(* IEC 61131-3 sources: manufacturing_io/scenes, 18 files *)

(* ---- a-to-b.st ---- *)
VAR
	START_EDGE : BOOL;
	PB_START_LAST : BOOL;
	STOP_REQ : BOOL;
	SEL_LAST : BOOL := TRUE;
	SEL_CHANGED : BOOL;
	T_DWELL : TON;
	T_WD : TON;
	EM_LAST : UDINT;
	STEP_LAST : UDINT;
	GONE : UDINT;
	MEM_CV : BOOL;
	IND_CV_LAST : BOOL;
	ESTOP : BOOL;
	READY : BOOL;
	MASTER_ON : BOOL;
	HOMED : BOOL;
	MASTER_EDGE : BOOL;
	PB_MASTER_LAST : BOOL;
	HOME_EDGE : BOOL;
	PB_HOME_LAST : BOOL;
END_VAR
// a-to-b: load one part, carry it to the end sensor, dwell, discharge it to the unloader, repeat
// until STOP. The same sequence runs without a PLC in a-to-b.ctl.js.
//
// Waiting steps wait for an INVARIANT, not for a counter to move: a change cannot say which
// part moved (measured on the simulator: parts piled up, then pipelined).
//
// The panel has a selector AUTO / INDIVIDUAL (rb4axis): START only in AUTO, the individual buttons
// only in INDIVIDUAL, and a change while the sequence runs is a FAULT, not a pause.

START_EDGE := PB_START AND NOT PB_START_LAST;
PB_START_LAST := PB_START;
IF PB_CSTOP THEN
	STOP_REQ := TRUE;
END_IF;
SEL_CHANGED := SEL_AUTO <> SEL_LAST;
SEL_LAST := SEL_AUTO;

// The master circuit, as on the cell panel: E-STOP is a latching mushroom, MASTER ON energises
// the machine, and nothing runs without it. An E-STOP also loses the home position.
ESTOP := PB_ESTOP;
MASTER_EDGE := PB_MASTER AND NOT PB_MASTER_LAST;
PB_MASTER_LAST := PB_MASTER;
HOME_EDGE := PB_HOME AND NOT PB_HOME_LAST;
PB_HOME_LAST := PB_HOME;
IF ESTOP THEN
	MASTER_ON := FALSE;
	HOMED := FALSE;
ELSIF MASTER_EDGE THEN
	MASTER_ON := TRUE;
END_IF;
READY := MASTER_ON AND NOT ESTOP;

// A write-off goes STALE when the part turns up after all - the hand puts it back, or it reaches
// the unloader later. Then RM + GONE runs PAST EM and step 40 stops waiting at all. GONE is a
// UDINT, so EM1_CNT - RM1_CNT with RM ahead underflows to about 4 billion: guard before you
// subtract.
IF RM1_CNT >= EM1_CNT THEN
	GONE := 0;
ELSIF RM1_CNT + GONE > EM1_CNT THEN
	GONE := EM1_CNT - RM1_CNT;
END_IF;

CASE ST1_STEP OF
	0:	// idle
		CV1_RUN := FALSE;
		EM1_EMIT := FALSE;
		IF START_EDGE AND SEL_AUTO AND READY AND HOMED THEN
			STOP_REQ := FALSE;
			EM_LAST := EM1_CNT;
			ST1_STEP := 10;
		END_IF;
	10:	// load one part: the command is held until the loader's counter answers it
		EM1_EMIT := TRUE;
		IF EM1_CNT <> EM_LAST THEN
			EM1_EMIT := FALSE;
			ST1_STEP := 15;
		END_IF;
	15:	// the beam must be clear before this part runs to it
		CV1_RUN := TRUE;
		IF NOT PE_END THEN
			ST1_STEP := 20;
		END_IF;
	20:	// carry it to the end sensor
		CV1_RUN := TRUE;
		IF PE_END THEN
			CV1_RUN := FALSE;
			ST1_STEP := 30;
		END_IF;
	30:	// dwell
		IF T_DWELL.Q THEN
			ST1_STEP := 40;
		END_IF;
	40:	// discharge: every part loaded has left the belt (counting the write-offs)
		CV1_RUN := TRUE;
		IF RM1_CNT + GONE >= EM1_CNT THEN
			CV1_RUN := FALSE;
			ST1_STEP := 50;
		END_IF;
	50:	// cycle complete
		CYCLE_CNT := CYCLE_CNT + 1;
		IF STOP_REQ THEN
			ST1_STEP := 0;
		ELSE
			EM_LAST := EM1_CNT;
			ST1_STEP := 10;
		END_IF;
	800:	// HOME: nothing here is positioned, so home only has to leave the line quiet
		CV1_RUN := FALSE;
		EM1_EMIT := FALSE;
		HOMED := TRUE;
		ST1_STEP := 0;
	910:	// E-STOP: the master circuit is open, so every solenoid de-energises - which is what
		// really happens: a 5/2 single-solenoid valve springs back, a double one holds.
		CV1_RUN := FALSE;
		EM1_EMIT := FALSE;
		IF READY THEN	// MASTER ON after the mushroom is released
			ST1_STEP := 0;
		END_IF;
	900:	// FAULT: a step stopped moving. Hold everything until START acknowledges it.
		CV1_RUN := FALSE;
		EM1_EMIT := FALSE;
		IF START_EDGE AND SEL_AUTO THEN
			STOP_REQ := FALSE;
			// Acknowledging writes off whatever never reached the unloader. Only HERE: at every
			// START it would write off parts still legitimately on the belt, and then an older
			// part's removal ends this cycle - the pipelining bug that cost two live rounds.
			GONE := EM1_CNT - RM1_CNT;
			ST1_STEP := 0;
		END_IF;
END_CASE;

T_DWELL(In := (ST1_STEP = 30), PT := T#500ms);

// Watchdog: a running step that stops moving is a jam, not patience. A selector change while
// running trips the same way.
T_WD(In := (ST1_STEP = STEP_LAST) AND (ST1_STEP <> 0) AND (ST1_STEP <> 900) AND (ST1_STEP <> 910), PT := T#15s);
IF ST1_STEP <> STEP_LAST THEN
	STEP_LAST := ST1_STEP;
END_IF;
IF T_WD.Q OR (SEL_CHANGED AND (ST1_STEP <> 0) AND (ST1_STEP <> 900) AND (ST1_STEP <> 910)) THEN
	ST1_STEP := 900;
	CV1_RUN := FALSE;
	EM1_EMIT := FALSE;
END_IF;

// E-STOP at any moment, and the HOME button when the machine is energised and idle.
IF ESTOP THEN
	IF ST1_STEP <> 910 THEN
		ST1_STEP := 910;
	END_IF;
	CV1_RUN := FALSE;
	EM1_EMIT := FALSE;
ELSIF HOME_EDGE AND READY AND (ST1_STEP = 0) THEN
	ST1_STEP := 800;
END_IF;

AUTO_RUN := (ST1_STEP <> 0) AND (ST1_STEP <> 800) AND (ST1_STEP <> 900) AND (ST1_STEP <> 910);

// Individual operation: the buttons are momentary; the PLC keeps a toggle
// memory per actuator and clears it when INDIVIDUAL ends, so nothing stays latched into AUTO.
IF NOT SEL_AUTO AND NOT AUTO_RUN AND READY AND (ST1_STEP <> 800) THEN
	IF IND_CV AND NOT IND_CV_LAST THEN
		MEM_CV := NOT MEM_CV;
	END_IF;
	CV1_RUN := MEM_CV;
	EM1_EMIT := IND_FEED;
ELSE
	MEM_CV := FALSE;
END_IF;
IND_CV_LAST := IND_CV;

// The speed override the operator dialled in, passed on to the axes and the belts.
OVR := OVR_SET;

PL_START := AUTO_RUN;
PL_MASTER := MASTER_ON;
PL_HOME := HOMED;

(* ---- assembler.st ---- *)
VAR
	START_EDGE : BOOL;
	PB_START_LAST : BOOL;
	STOP_REQ : BOOL;
	EM_B_LAST : UDINT;
	EM_L_LAST : UDINT;
	NEXT_ST : INT;
	T_PRESS : TON;
END_VAR
// assembler: a 4-station cam indexer. Every station works during the same dwell - load a base,
// drop a lid on it, press it - and then the table turns one step, carrying each assembly to the
// next station. The unload station simply takes whatever reaches it. The same sequence runs
// without a PLC in assembler.ctl.js.
//
// The index waits for an INVARIANT, TBL_STATION = NEXT_ST, not for the station to change: a
// change cannot say which index it belonged to, and OPC UA sampling can miss a short state.
// Each feeder command is held until that feeder's own counter answers it.

START_EDGE := PB_START AND NOT PB_START_LAST;
PB_START_LAST := PB_START;
IF PB_STOP THEN
	STOP_REQ := TRUE;
END_IF;

CASE ST1_STEP OF
	0:	// idle, table stopped in a dwell, press up
		TBL_RUN := FALSE;
		EM_B_EMIT := FALSE;
		EM_L_EMIT := FALSE;
		SOL_PRESS_DN := FALSE;
		SOL_PRESS_UP := TRUE;
		IF START_EDGE AND TBL_INPOS AND AS_PRESS_UP THEN
			STOP_REQ := FALSE;
			EM_B_LAST := EM_B_CNT;
			ST1_STEP := 10;
		END_IF;
	10:	// station 0: load a base into the nest
		EM_B_EMIT := TRUE;
		IF EM_B_CNT <> EM_B_LAST THEN
			EM_B_EMIT := FALSE;
			EM_L_LAST := EM_L_CNT;
			ST1_STEP := 20;
		END_IF;
	20:	// station 1: drop a lid onto the base that arrived there
		EM_L_EMIT := TRUE;
		IF EM_L_CNT <> EM_L_LAST THEN
			EM_L_EMIT := FALSE;
			ST1_STEP := 30;
		END_IF;
	30:	// station 2: press down
		SOL_PRESS_UP := FALSE;
		SOL_PRESS_DN := TRUE;
		IF AS_PRESS_DN THEN
			ST1_STEP := 40;
		END_IF;
	40:	// hold the press on the lid
		IF T_PRESS.Q THEN
			ST1_STEP := 50;
		END_IF;
	50:	// press up, and pick the station this index must reach
		SOL_PRESS_DN := FALSE;
		SOL_PRESS_UP := TRUE;
		IF AS_PRESS_UP THEN
			NEXT_ST := (TBL_STATION + 1) MOD 4;
			ST1_STEP := 60;
		END_IF;
	60:	// turn the table one station
		TBL_RUN := TRUE;
		IF TBL_INPOS AND TBL_STATION = NEXT_ST THEN
			TBL_RUN := FALSE;
			CYCLE_CNT := CYCLE_CNT + 1;
			IF STOP_REQ THEN
				ST1_STEP := 0;
			ELSE
				EM_B_LAST := EM_B_CNT;
				ST1_STEP := 10;
			END_IF;
		END_IF;
END_CASE;

T_PRESS(In := (ST1_STEP = 40), PT := T#300ms);
AUTO_RUN := ST1_STEP <> 0;
PL_START := AUTO_RUN;

(* ---- blurobot.st ---- *)
VAR
	START_EDGE : BOOL;
	PB_START_LAST : BOOL;
	STOP_REQ : BOOL;
	T_WD : TON;
	T_GRIP : TON;
	STEP_LAST : UDINT;
	i : INT;
	j : INT;
	SRC : INT;
	DST : INT;
	IDX : INT;
	HOLDING : BOOL;
	AT_POSE : BOOL;
	CLEARED : BOOL;
	RAIL_X : LREAL;
	ARM_AT_1 : LREAL;
	ARM_AT_2 : LREAL;
	ARM_AT_3 : LREAL;
	ARM_UP_1 : LREAL;
	ARM_UP_2 : LREAL;
	ARM_UP_3 : LREAL;
	COVER_OK : BOOL;
	IN_ZONE : BOOL;
	SHUT : BOOL;
	// What the PLC BELIEVES about each station, and each machine's own clock. These are program
	// variables, not machine IO: nothing in the plant senses them. rb4axis keeps the same values in
	// SIM_ST_STATE / SIM_ST_TIMER and only publishes them so its viewer can draw the cell.
	//   0 empty, 1 processing, 2 finished and waiting to be collected
	ICC1_STATE : INT;
	ICC2_STATE : INT;
	DW1_STATE : INT;
	DW2_STATE : INT;
	ICC1_TIMER : LREAL;
	ICC2_TIMER : LREAL;
	DW1_TIMER : LREAL;
	DW2_TIMER : LREAL;
	// The cover target each station is latched on. Execute is LATCHED on its rising edge, like
	// every other axis here, so holding it true from the first scan means the target is never
	// re-read: measured, the covers held their startup 80 while the target sat at 0, no ICC clock
	// ever ran, and no board ever finished. A change re-pulses Execute.
	ICC1_CV_WANT : LREAL;
	ICC2_CV_WANT : LREAL;
	DW1_CV_WANT : LREAL;
	DW2_CV_WANT : LREAL;
END_VAR
// blurobot - a PORT of rb4axis PRG_SIM_ROBOT.st. The cell, the station table, the job priorities,
// the step numbers and the timings are that program's; only the tag shape differs, because this
// repo binds scalar tags while the original keeps SIM_ST_* arrays.
//
//   station   type  rail x   surface z   process
//   WIP IN     0     -1400      250        -      stock is not simulated: always FULL
//   ICC 1      1      -700      285      17.0 s   test; the cover presses the PCB onto the probes
//   ICC 2      1      -300      285      17.0 s
//   DW 1       2       300      250      15.0 s   data writer
//   DW 2       2       700      250      15.0 s
//   WIP OUT    3      1400      250        -      the product leaves: always EMPTY
//
// Job priority, and the ORDER is the behaviour:
//   1. fill an EMPTY ICC from WIP IN - both - before anything else. That is what buffer means: the
//      17 s tester must not idle while the robot runs errands for DW.
//   2. empty a FINISHED DW to WIP OUT, ahead of 3, so a free DW always exists. Without it two full
//      DWs plus two finished ICCs deadlock, and the deadlock looks like a robot that stopped.
//   3. move a FINISHED ICC to an EMPTY DW.
//
// Poses were measured against the scene's own kinematics with the carriage at z 200: all twelve
// (six surfaces + six 140 mm approaches) solve with 67.3 deg of worst-case joint margin. Only two
// station heights exist, so there are four arm poses and the rail carries the difference.
//
// Execute is a LEVEL held until every axis reports Done, and the next move waits for Done to fall
// again: a one-scan pulse falls between two OPC UA samples.

START_EDGE := PB_START AND NOT PB_START_LAST;
PB_START_LAST := PB_START;
IF PB_STOP THEN
	STOP_REQ := TRUE;
END_IF;

AT_POSE := A0_DONE AND A1_DONE AND A2_DONE AND A3_DONE;
CLEARED := NOT A0_DONE AND NOT A1_DONE AND NOT A2_DONE AND NOT A3_DONE;

// ---------------------------------------------------------------- the machines
// Each keeps its OWN timer, running together: that is the whole point of a buffer, ICC 1 and ICC 2
// must be able to test at the same time while the robot is away. The clock runs ONLY with the
// cover shut - the cover presses the PCB onto the probes, and counting before it closes means
// claiming a test on a board nothing has touched.
//
// The cover closes only while processing and REOPENS if the arm is in its sweep: a light curtain,
// not a delay. Without it the leaf swings onto an arm that is still lifting out.
IN_ZONE := (ABS(A0_POS - (-700.0)) < 200.0) AND (A1_POS < 60.0);
SHUT := (ICC1_STATE = 1) AND NOT IN_ZONE;
IF SHUT THEN COVER_TARGET := 0.0; ELSE COVER_TARGET := 80.0; END_IF;
IF COVER_TARGET <> ICC1_CV_WANT THEN
	ICC1_CV_WANT := COVER_TARGET;
	ICC1_CV_EXEC := FALSE;
ELSE
	ICC1_CV_TGT := COVER_TARGET;
	ICC1_CV_EXEC := TRUE;
END_IF;
IF (ICC1_STATE = 1) AND (ICC1_CV_POS <= 0.5) THEN
	ICC1_TIMER := ICC1_TIMER - 0.002;
	IF ICC1_TIMER <= 0.0 THEN ICC1_TIMER := 0.0; ICC1_STATE := 2; END_IF;
END_IF;

IN_ZONE := (ABS(A0_POS - (-300.0)) < 200.0) AND (A1_POS < 60.0);
SHUT := (ICC2_STATE = 1) AND NOT IN_ZONE;
IF SHUT THEN COVER_TARGET := 0.0; ELSE COVER_TARGET := 80.0; END_IF;
IF COVER_TARGET <> ICC2_CV_WANT THEN
	ICC2_CV_WANT := COVER_TARGET;
	ICC2_CV_EXEC := FALSE;
ELSE
	ICC2_CV_TGT := COVER_TARGET;
	ICC2_CV_EXEC := TRUE;
END_IF;
IF (ICC2_STATE = 1) AND (ICC2_CV_POS <= 0.5) THEN
	ICC2_TIMER := ICC2_TIMER - 0.002;
	IF ICC2_TIMER <= 0.0 THEN ICC2_TIMER := 0.0; ICC2_STATE := 2; END_IF;
END_IF;

IN_ZONE := (ABS(A0_POS - 300.0) < 200.0) AND (A1_POS < 60.0);
SHUT := (DW1_STATE = 1) AND NOT IN_ZONE;
IF SHUT THEN COVER_TARGET := 0.0; ELSE COVER_TARGET := 80.0; END_IF;
IF COVER_TARGET <> DW1_CV_WANT THEN
	DW1_CV_WANT := COVER_TARGET;
	DW1_CV_EXEC := FALSE;
ELSE
	DW1_CV_TGT := COVER_TARGET;
	DW1_CV_EXEC := TRUE;
END_IF;
IF (DW1_STATE = 1) AND (DW1_CV_POS <= 0.5) THEN
	DW1_TIMER := DW1_TIMER - 0.002;
	IF DW1_TIMER <= 0.0 THEN DW1_TIMER := 0.0; DW1_STATE := 2; END_IF;
END_IF;

IN_ZONE := (ABS(A0_POS - 700.0) < 200.0) AND (A1_POS < 60.0);
SHUT := (DW2_STATE = 1) AND NOT IN_ZONE;
IF SHUT THEN COVER_TARGET := 0.0; ELSE COVER_TARGET := 80.0; END_IF;
IF COVER_TARGET <> DW2_CV_WANT THEN
	DW2_CV_WANT := COVER_TARGET;
	DW2_CV_EXEC := FALSE;
ELSE
	DW2_CV_TGT := COVER_TARGET;
	DW2_CV_EXEC := TRUE;
END_IF;
IF (DW2_STATE = 1) AND (DW2_CV_POS <= 0.5) THEN
	DW2_TIMER := DW2_TIMER - 0.002;
	IF DW2_TIMER <= 0.0 THEN DW2_TIMER := 0.0; DW2_STATE := 2; END_IF;
END_IF;

// WIP IN never runs out and WIP OUT never fills up: the stock either side of the cell is not
// simulated, and pretending otherwise would starve or block a cell that never does either. Those
// two need no state variable at all - the job selection below simply treats them that way.

// ---------------------------------------------------------- the pose for IDX
// Four arm poses only, because the six stations sit at just two heights; the rail carries the
// rest. Measured against the scene's own kinematics with the carriage at z 200.
CASE IDX OF
	0:	RAIL_X := -1400.0;
	1:	RAIL_X := -700.0;
	2:	RAIL_X := -300.0;
	3:	RAIL_X := 300.0;
	4:	RAIL_X := 700.0;
	5:	RAIL_X := 1400.0;
ELSE
	RAIL_X := 0.0;
END_CASE;

IF (IDX = 1) OR (IDX = 2) THEN
	// the 285 mm tables
	ARM_AT_1 := 15.72;   ARM_AT_2 := -71.33;   ARM_AT_3 := -34.39;
	ARM_UP_1 := 36.55;   ARM_UP_2 := -77.44;   ARM_UP_3 := -49.11;
ELSE
	// the 250 mm tables
	ARM_AT_1 := 9.76;   ARM_AT_2 := -67.25;   ARM_AT_3 := -32.5;
	ARM_UP_1 := 31.86;   ARM_UP_2 := -77.37;   ARM_UP_3 := -44.49;
END_IF;

// The WIP racks are open - no cover, so nothing to wait for.
CASE IDX OF
	1:	COVER_OK := ICC1_CV_POS >= 79.5;
	2:	COVER_OK := ICC2_CV_POS >= 79.5;
	3:	COVER_OK := DW1_CV_POS >= 79.5;
	4:	COVER_OK := DW2_CV_POS >= 79.5;
ELSE
	COVER_OK := TRUE;
END_CASE;

// ------------------------------------------------- every station holds what is on it
// Only the one being picked from lets go, and only while the gripper takes the board. Measured
// with no clamp set at all: the nest held nothing, WIPIN_P never came true, and the fingers closed
// to zero straight through the PCB - a part's width is only measured for a FREE part, so gripping
// a still-held board reads as gripping air and the closed switch asserts for the wrong reason.
// WIP IN is an ENDLESS stock: the PLC pins its state to "full" because the racks either side of
// the cell are not simulated, so the plant has to keep a board there or the cell runs dry and the
// next grip closes on air. A LEVEL held until the feeder's own count answers it, never a pulse,
// and only while that nest is empty and the arm is not taking from it.
EM_IN_EMIT := NOT WIPIN_P AND NOT (((ST1_STEP = 14) OR (ST1_STEP = 15)) AND (IDX = 0));

WIPIN_CLAMP := NOT (((ST1_STEP = 14) OR (ST1_STEP = 15)) AND (IDX = 0));
ICC1_CLAMP := NOT (((ST1_STEP = 14) OR (ST1_STEP = 15)) AND (IDX = 1));
ICC2_CLAMP := NOT (((ST1_STEP = 14) OR (ST1_STEP = 15)) AND (IDX = 2));
DW1_CLAMP := NOT (((ST1_STEP = 14) OR (ST1_STEP = 15)) AND (IDX = 3));
DW2_CLAMP := NOT (((ST1_STEP = 14) OR (ST1_STEP = 15)) AND (IDX = 4));
WIPOUT_CLAMP := NOT (((ST1_STEP = 14) OR (ST1_STEP = 15)) AND (IDX = 5));

CASE ST1_STEP OF
	0:	// pick a job - the order of these three searches IS the cell's behaviour
		SRC := -1;
		DST := -1;
		IF (ICC1_STATE = 0) THEN SRC := 0; DST := 1; END_IF;
		IF (DST < 0) AND (ICC2_STATE = 0) THEN SRC := 0; DST := 2; END_IF;
		IF (DST < 0) AND (DW1_STATE = 2) THEN SRC := 3; DST := 5; END_IF;
		IF (DST < 0) AND (DW2_STATE = 2) THEN SRC := 4; DST := 5; END_IF;
		IF (DST < 0) AND (ICC1_STATE = 2) AND (DW1_STATE = 0) THEN SRC := 1; DST := 3; END_IF;
		IF (DST < 0) AND (ICC1_STATE = 2) AND (DW2_STATE = 0) THEN SRC := 1; DST := 4; END_IF;
		IF (DST < 0) AND (ICC2_STATE = 2) AND (DW1_STATE = 0) THEN SRC := 2; DST := 3; END_IF;
		IF (DST < 0) AND (ICC2_STATE = 2) AND (DW2_STATE = 0) THEN SRC := 2; DST := 4; END_IF;
		IF DST >= 0 THEN
			IDX := SRC;
			ST1_STEP := 5;
		ELSIF STOP_REQ THEN
			STOP_REQ := FALSE;
		END_IF;

	5:	// fold to the travel pose - axes 1-3 only, the rail is not touched
		A1_TGT := 90.0;   A2_TGT := -90.0;   A3_TGT := -90.0;
		A1_EXEC := TRUE;   A2_EXEC := TRUE;   A3_EXEC := TRUE;
		IF A1_DONE AND A2_DONE AND A3_DONE THEN
			ST1_STEP := 7;
		END_IF;

	7:	// slide the rail. The arm MUST be folded: travelling while reaching down sweeps every
		// machine it passes, and on screen that looks perfectly smooth.
		A0_TGT := RAIL_X;
		A0_EXEC := TRUE;
		ST1_STEP := 8;

	8:	// TWO things, and the wait is HERE rather than after the approach is asked for: asking
		// while the cover is still shut gets the move refused, nothing moves, and Done stays TRUE -
		// so the next step would drive straight down from the travel pose, skipping the approach.
		IF A0_DONE AND COVER_OK THEN
			ST1_STEP := 10;
		END_IF;

	10:	// above the station
		A0_TGT := RAIL_X;   A1_TGT := ARM_UP_1;   A2_TGT := ARM_UP_2;   A3_TGT := ARM_UP_3;
		A0_EXEC := TRUE;   A1_EXEC := TRUE;   A2_EXEC := TRUE;   A3_EXEC := TRUE;
		IF AT_POSE THEN ST1_STEP := 11; END_IF;
	11:	A0_EXEC := FALSE; A1_EXEC := FALSE; A2_EXEC := FALSE; A3_EXEC := FALSE;
		IF CLEARED THEN ST1_STEP := 12; END_IF;

	12:	// straight down onto the surface - the gripper pinches from ABOVE
		A0_TGT := RAIL_X;   A1_TGT := ARM_AT_1;   A2_TGT := ARM_AT_2;   A3_TGT := ARM_AT_3;
		A0_EXEC := TRUE;   A1_EXEC := TRUE;   A2_EXEC := TRUE;   A3_EXEC := TRUE;
		IF AT_POSE THEN ST1_STEP := 13; END_IF;
	13:	A0_EXEC := FALSE; A1_EXEC := FALSE; A2_EXEC := FALSE; A3_EXEC := FALSE;
		IF CLEARED THEN ST1_STEP := 14; END_IF;

	14:	// the station let go above; close on the board
		GRIP_CLOSE := TRUE;
		ST1_STEP := 15;

	15:	// NOT GRIP_CLOSED: that switch sits at FULL close, and a good grip STOPS at the product
		// width - measured, the jaws ran 90 -> 60 mm half-opening on a 120 mm board and held
		// there. Waiting for GRIP_CLOSED waits for the signal that means the fingers found
		// NOTHING (rb4axis SIM_GRIP_TUTUP). Confirm on the open switch dropping and staying
		// dropped, so a board slipping out of the fingers restarts the confirm.
		IF T_GRIP.Q THEN
			HOLDING := TRUE;
			// the machine it came OUT of is empty now - SRC, never IDX; WIP IN is never emptied
			IF SRC = 1 THEN ICC1_STATE := 0; END_IF;
			IF SRC = 2 THEN ICC2_STATE := 0; END_IF;
			IF SRC = 3 THEN DW1_STATE := 0; END_IF;
			IF SRC = 4 THEN DW2_STATE := 0; END_IF;
			ST1_STEP := 16;
		END_IF;

	16:	A0_TGT := RAIL_X;   A1_TGT := ARM_UP_1;   A2_TGT := ARM_UP_2;   A3_TGT := ARM_UP_3;
		A0_EXEC := TRUE;   A1_EXEC := TRUE;   A2_EXEC := TRUE;   A3_EXEC := TRUE;
		IF AT_POSE THEN ST1_STEP := 17; END_IF;
	17:	A0_EXEC := FALSE; A1_EXEC := FALSE; A2_EXEC := FALSE; A3_EXEC := FALSE;
		IF CLEARED THEN ST1_STEP := 18; END_IF;

	18:	A1_TGT := 90.0;   A2_TGT := -90.0;   A3_TGT := -90.0;
		A1_EXEC := TRUE;   A2_EXEC := TRUE;   A3_EXEC := TRUE;
		IF A1_DONE AND A2_DONE AND A3_DONE THEN
			IDX := DST;
			ST1_STEP := 20;
		END_IF;

	20:	A0_TGT := RAIL_X;
		A0_EXEC := TRUE;
		ST1_STEP := 21;

	21:	// same as step 8: the destination cover must be open BEFORE the approach is asked for
		IF A0_DONE AND COVER_OK THEN
			ST1_STEP := 22;
		END_IF;

	22:	A0_TGT := RAIL_X;   A1_TGT := ARM_UP_1;   A2_TGT := ARM_UP_2;   A3_TGT := ARM_UP_3;
		A0_EXEC := TRUE;   A1_EXEC := TRUE;   A2_EXEC := TRUE;   A3_EXEC := TRUE;
		IF AT_POSE THEN ST1_STEP := 23; END_IF;
	23:	A0_EXEC := FALSE; A1_EXEC := FALSE; A2_EXEC := FALSE; A3_EXEC := FALSE;
		IF CLEARED THEN ST1_STEP := 24; END_IF;

	24:	A0_TGT := RAIL_X;   A1_TGT := ARM_AT_1;   A2_TGT := ARM_AT_2;   A3_TGT := ARM_AT_3;
		A0_EXEC := TRUE;   A1_EXEC := TRUE;   A2_EXEC := TRUE;   A3_EXEC := TRUE;
		IF AT_POSE THEN ST1_STEP := 25; END_IF;
	25:	A0_EXEC := FALSE; A1_EXEC := FALSE; A2_EXEC := FALSE; A3_EXEC := FALSE;
		IF CLEARED THEN ST1_STEP := 26; END_IF;

	26:	GRIP_CLOSE := FALSE;
		ST1_STEP := 27;

	27:	IF GRIP_OPEN THEN
			HOLDING := FALSE;
			// WIP OUT: the product leaves the cell, and THAT is where cycle time is taken -
			// exit to exit, because that is what decides how many boards an hour leave.
			// Written against DST, never IDX: IDX is reused for source then destination, so on a
			// job whose SOURCE was this same station the step-15 clear would zero the state just
			// set here. Measured: ICC 1 was loaded, set to processing, then reported empty again,
			// so its cover never shut and its 17 s clock never ran.
			IF DST = 5 THEN
				CYCLE_CNT := CYCLE_CNT + 1;
			ELSE
				// the station starts its own clock; each runs independently
				IF DST = 1 THEN ICC1_STATE := 1; ICC1_TIMER := 17.0; END_IF;
				IF DST = 2 THEN ICC2_STATE := 1; ICC2_TIMER := 17.0; END_IF;
				IF DST = 3 THEN DW1_STATE := 1; DW1_TIMER := 15.0; END_IF;
				IF DST = 4 THEN DW2_STATE := 1; DW2_TIMER := 15.0; END_IF;
			END_IF;
			ST1_STEP := 28;
		END_IF;

	28:	A0_TGT := RAIL_X;   A1_TGT := ARM_UP_1;   A2_TGT := ARM_UP_2;   A3_TGT := ARM_UP_3;
		A0_EXEC := TRUE;   A1_EXEC := TRUE;   A2_EXEC := TRUE;   A3_EXEC := TRUE;
		IF AT_POSE THEN ST1_STEP := 29; END_IF;
	29:	A0_EXEC := FALSE; A1_EXEC := FALSE; A2_EXEC := FALSE; A3_EXEC := FALSE;
		IF CLEARED THEN ST1_STEP := 30; END_IF;

	30:	A1_TGT := 90.0;   A2_TGT := -90.0;   A3_TGT := -90.0;
		A1_EXEC := TRUE;   A2_EXEC := TRUE;   A3_EXEC := TRUE;
		IF A1_DONE AND A2_DONE AND A3_DONE THEN
			ST1_STEP := 31;
		END_IF;

	31:	// Cycle stop is served HERE: the product is placed and the arm folded, so stopping is
		// controlled and START works again straight away.
		IF STOP_REQ THEN
			STOP_REQ := FALSE;
		END_IF;
		ST1_STEP := 0;

	900:	// FAULT: a step stopped moving. Hold everything, and KEEP the grip - a real arm does
		// not open its fingers over the floor.
		A0_EXEC := FALSE; A1_EXEC := FALSE; A2_EXEC := FALSE; A3_EXEC := FALSE;
		IF START_EDGE THEN
			STOP_REQ := FALSE;
			ST1_STEP := 0;
		END_IF;
END_CASE;

// The grip confirm: fingers off the open switch and staying off for 300 ms.
T_GRIP(In := (ST1_STEP = 15) AND GRIP_CLOSE AND NOT GRIP_OPEN, PT := T#300ms);

// Watchdog. 30 s, not 15: a station's own process is 17 s, and the arm legitimately waits at step
// 8 and 21 for a cover that only opens once that test has finished.
T_WD(In := (ST1_STEP = STEP_LAST) AND (ST1_STEP <> 0) AND (ST1_STEP <> 900), PT := T#30s);
IF ST1_STEP <> STEP_LAST THEN
	STEP_LAST := ST1_STEP;
END_IF;
IF T_WD.Q THEN
	ST1_STEP := 900;
	A0_EXEC := FALSE; A1_EXEC := FALSE; A2_EXEC := FALSE; A3_EXEC := FALSE;
END_IF;

AUTO_RUN := (ST1_STEP <> 0) AND (ST1_STEP <> 900);
PL_START := AUTO_RUN;

(* ---- buffer-queue.st ---- *)
VAR
	START_EDGE : BOOL;
	PB_START_LAST : BOOL;
	STOP_REQ : BOOL;
	SEL_LAST : BOOL := TRUE;
	SEL_CHANGED : BOOL;
	EM_LAST : UDINT;
	T_SETTLE : TON;
	T_DEMAND : TON;
	T_WD : TON;
	STEP_LAST : UDINT;
	GONE : UDINT;
	MEM_CV : BOOL;
	IND_CV_LAST : BOOL;
	MEM_HOLD : BOOL;
	IND_HOLD_LAST : BOOL;
	MEM_GATE : BOOL;
	IND_GATE_LAST : BOOL;
	ESTOP : BOOL;
	READY : BOOL;
	MASTER_ON : BOOL;
	HOMED : BOOL;
	MASTER_EDGE : BOOL;
	PB_MASTER_LAST : BOOL;
	HOME_EDGE : BOOL;
	PB_HOME_LAST : BOOL;
END_VAR
// buffer-queue: a stop-and-go escapement. Two stopper cylinders stand 300 mm apart over the belt:
// the HOLD pin meters parts into the pocket between them, the GATE pin holds the metered part
// until the downstream station asks for it. Each pin has its own up and down reed switches, and
// each position has its own photo-eye. The same sequence runs without a PLC in buffer-queue.ctl.js.
//
// ONE part is in the line at a time, and that is not a simplification: a pin cannot come down
// between parts that TOUCH, so an escapement can only work where the parts arrive with a gap
// (measured, tests/rapier.test.js). The loader is therefore metered by the sequence, and the
// HOLD pin always comes down on free belt.
//
// The panel has a selector AUTO / INDIVIDUAL: START only in AUTO, the individual buttons only in
// INDIVIDUAL, and a change while the sequence runs is a FAULT, not a pause.

START_EDGE := PB_START AND NOT PB_START_LAST;
PB_START_LAST := PB_START;
IF PB_CSTOP THEN
	STOP_REQ := TRUE;
END_IF;
SEL_CHANGED := SEL_AUTO <> SEL_LAST;
SEL_LAST := SEL_AUTO;

// The master circuit, as on the cell panel: E-STOP is a latching mushroom, MASTER ON energises
// the machine, and nothing runs without it. An E-STOP also loses the home position.
ESTOP := PB_ESTOP;
MASTER_EDGE := PB_MASTER AND NOT PB_MASTER_LAST;
PB_MASTER_LAST := PB_MASTER;
HOME_EDGE := PB_HOME AND NOT PB_HOME_LAST;
PB_HOME_LAST := PB_HOME;
IF ESTOP THEN
	MASTER_ON := FALSE;
	HOMED := FALSE;
ELSIF MASTER_EDGE THEN
	MASTER_ON := TRUE;
END_IF;
READY := MASTER_ON AND NOT ESTOP;

// A write-off goes STALE when the part turns up after all, and then RM + GONE runs PAST EM and
// the step waiting on that invariant stops waiting at all. GONE is a UDINT, so the subtraction
// underflows to about 4 billion when RM is ahead: guard before you subtract.
IF RM_CNT >= EM_CNT THEN
	GONE := 0;
ELSIF RM_CNT + GONE > EM_CNT THEN
	GONE := EM_CNT - RM_CNT;
END_IF;
CASE ST1_STEP OF
	0:	// idle: belt off, both pins retracted
		CV_RUN := FALSE;
		EM_EMIT := FALSE;
		SOL_HOLD := FALSE;
		SOL_GATE := FALSE;
		IF START_EDGE AND SEL_AUTO AND READY AND HOMED AND AS_HOLD_UP AND AS_GATE_UP THEN
			STOP_REQ := FALSE;
			ST1_STEP := 10;
		END_IF;
	10:	// belt on, and the gate pin goes down first: nothing may leave until the escapement is armed
		CV_RUN := TRUE;
		SOL_GATE := TRUE;
		IF AS_GATE_DN THEN
			ST1_STEP := 15;
		END_IF;
	15:	// hold pin down: the line is now blocked at both ends
		SOL_HOLD := TRUE;
		IF AS_HOLD_DN THEN
			ST1_STEP := 20;
		END_IF;
	20:	// let one part into the line; the command is held until the loader's counter answers it
		EM_EMIT := TRUE;
		IF EM_CNT <> EM_LAST THEN
			EM_EMIT := FALSE;
			ST1_STEP := 25;
		END_IF;
	25:	// it runs down the belt to the hold pin
		IF PE_HOLD THEN
			ST1_STEP := 30;
		END_IF;
	30:	// let it settle against the pin
		IF T_SETTLE.Q THEN
			ST1_STEP := 40;
		END_IF;
	40:	// GO: the hold pin lifts and this one part runs into the pocket between the pins
		SOL_HOLD := FALSE;
		IF AS_HOLD_UP THEN
			ST1_STEP := 45;
		END_IF;
	45:	// wait until the part has cleared the hold eye
		IF NOT PE_HOLD THEN
			ST1_STEP := 50;
		END_IF;
	50:	// STOP: the pin comes down again on FREE BELT. It can only do that because the next part
		// has not been fed yet - a pin cannot land between parts that touch.
		SOL_HOLD := TRUE;
		IF AS_HOLD_DN THEN
			ST1_STEP := 60;
		END_IF;
	60:	// the part arrives at the gate pin
		IF PE_GATE THEN
			ST1_STEP := 70;
		END_IF;
	70:	// it waits in the pocket until the downstream station asks for it
		IF T_DEMAND.Q THEN
			ST1_STEP := 80;
		END_IF;
	80:	// the gate lifts and the part leaves the pocket
		SOL_GATE := FALSE;
		IF NOT PE_GATE THEN
			ST1_STEP := 90;
		END_IF;
	90:	// gate down again, ready for the next one
		SOL_GATE := TRUE;
		IF AS_GATE_DN THEN
			ST1_STEP := 95;
		END_IF;
	95:	// cycle complete once every part let in has left the belt
		IF RM_CNT + GONE >= EM_CNT THEN
			CYCLE_CNT := CYCLE_CNT + 1;
			IF STOP_REQ THEN
				ST1_STEP := 0;
			ELSE
				EM_LAST := EM_CNT;
				ST1_STEP := 20;
			END_IF;
		END_IF;
	800:	// HOME: both pins retracted, so the line is clear, and the belt is quiet
		CV_RUN := FALSE;
		EM_EMIT := FALSE;
		SOL_HOLD := FALSE;
		SOL_GATE := FALSE;
		IF AS_HOLD_UP AND AS_GATE_UP THEN
			HOMED := TRUE;
			ST1_STEP := 0;
		END_IF;
	900:	// FAULT: a step stopped moving (a part taken, jammed or lost), or the selector was
		// turned while running.
		CV_RUN := FALSE;
		EM_EMIT := FALSE;
		SOL_HOLD := FALSE;
		SOL_GATE := FALSE;
		IF START_EDGE AND SEL_AUTO THEN
			STOP_REQ := FALSE;
			// Acknowledging writes off whatever never reached the outfeed. Only HERE.
			GONE := EM_CNT - RM_CNT;
			ST1_STEP := 0;
		END_IF;
	910:	// E-STOP: the master circuit is open, so every solenoid de-energises - which is what
		// really happens: a 5/2 single-solenoid valve springs back, a double one holds.
		CV_RUN := FALSE;
		EM_EMIT := FALSE;
		SOL_HOLD := FALSE;
		SOL_GATE := FALSE;
		IF READY THEN	// MASTER ON after the mushroom is released
			ST1_STEP := 0;
		END_IF;
END_CASE;

T_SETTLE(In := (ST1_STEP = 30), PT := T#300ms);
T_DEMAND(In := (ST1_STEP = 70), PT := T#1500ms);

// Watchdog: a running step that stops moving is a jam, not patience. A selector change while
// running trips the same way.
T_WD(In := (ST1_STEP = STEP_LAST) AND (ST1_STEP <> 0) AND (ST1_STEP <> 900) AND (ST1_STEP <> 910), PT := T#15s);
IF ST1_STEP <> STEP_LAST THEN
	STEP_LAST := ST1_STEP;
END_IF;
IF T_WD.Q OR (SEL_CHANGED AND (ST1_STEP <> 0) AND (ST1_STEP <> 900) AND (ST1_STEP <> 910)) THEN
	ST1_STEP := 900;
	CV_RUN := FALSE;
	EM_EMIT := FALSE;
	SOL_HOLD := FALSE;
	SOL_GATE := FALSE;
END_IF;

// E-STOP at any moment, and the HOME button when the machine is energised and idle.
IF ESTOP THEN
	IF ST1_STEP <> 910 THEN
		ST1_STEP := 910;
	END_IF;
	CV_RUN := FALSE;
	EM_EMIT := FALSE;
	SOL_HOLD := FALSE;
	SOL_GATE := FALSE;
ELSIF HOME_EDGE AND READY AND (ST1_STEP = 0) THEN
	ST1_STEP := 800;
END_IF;

AUTO_RUN := (ST1_STEP <> 0) AND (ST1_STEP <> 800) AND (ST1_STEP <> 900) AND (ST1_STEP <> 910);

// Individual operation: momentary buttons, a PLC toggle memory per actuator, cleared when
// INDIVIDUAL ends. The feed button pulses one part.
IF NOT SEL_AUTO AND NOT AUTO_RUN AND READY AND (ST1_STEP <> 800) THEN
	IF IND_CV AND NOT IND_CV_LAST THEN
		MEM_CV := NOT MEM_CV;
	END_IF;
	IF IND_HOLD AND NOT IND_HOLD_LAST THEN
		MEM_HOLD := NOT MEM_HOLD;
	END_IF;
	IF IND_GATE AND NOT IND_GATE_LAST THEN
		MEM_GATE := NOT MEM_GATE;
	END_IF;
	CV_RUN := MEM_CV;
	EM_EMIT := IND_FEED;
	SOL_HOLD := MEM_HOLD;
	SOL_GATE := MEM_GATE;
ELSE
	MEM_CV := FALSE;
	MEM_HOLD := FALSE;
	MEM_GATE := FALSE;
END_IF;
IND_CV_LAST := IND_CV;
IND_HOLD_LAST := IND_HOLD;
IND_GATE_LAST := IND_GATE;

// The speed override the operator dialled in, passed on to the axes and the belts.
OVR := OVR_SET;

PL_START := AUTO_RUN;
PL_MASTER := MASTER_ON;
PL_HOME := HOMED;

(* ---- carton-sorter.st ---- *)
VAR
	START_EDGE : BOOL;
	PB_START_LAST : BOOL;
	STOP_REQ : BOOL;
	SEL_LAST : BOOL := TRUE;
	SEL_CHANGED : BOOL;
	T_DIV_A : TON;
	T_DIV_B : TON;
	T_WD2 : TON;
	T_WD3 : TON;
	STEP2_LAST : UDINT;
	STEP3_LAST : UDINT;
	RUNNING : BOOL;
	SCAN_EDGE : BOOL;
	PE_IN_LAST : BOOL;
	UP_A_EDGE : BOOL;
	PE_UP_A_LAST : BOOL;
	UP_B_EDGE : BOOL;
	PE_UP_B_LAST : BOOL;
	NEXT_DEST : UINT;
	DEST : UINT;
	QA : ARRAY[0..15] OF UINT;
	QA_H : UINT;
	QA_T : UINT;
	QA_N : UINT;
	QB : ARRAY[0..15] OF UINT;
	QB_H : UINT;
	QB_T : UINT;
	QB_N : UINT;
	MEM_CV : BOOL;
	MEM_FEED : BOOL;
	MEM_SPA : BOOL;
	MEM_SPB : BOOL;
	IND_CV_LAST : BOOL;
	IND_FEED_LAST : BOOL;
	IND_SPA_LAST : BOOL;
	IND_SPB_LAST : BOOL;
	IND_ACTIVE : BOOL;
	ESTOP : BOOL;
	READY : BOOL;
	MASTER_ON : BOOL;
	HOMED : BOOL;
	MASTER_EDGE : BOOL;
	PB_MASTER_LAST : BOOL;
	HOME_EDGE : BOOL;
	PB_HOME_LAST : BOOL;
END_VAR
// carton-sorter: a sortation line on the Open Industry Project's own numbers - a 1.524 m belt at
// 2 m/s, cartons 600 x 400 x 400 at 10 kg fed 45 a minute, and two swing-blade diverters whose
// 2.127 m blade sweeps 1504 mm across the belt at 45 degrees, the belt itself driving the carton
// along the blade and onto a take-away at 1 m/s. The same sequence runs without a PLC in
// carton-sorter.ctl.js - keep the two in step.
//
// TRACKING is the whole job here, and it is a SHIFT REGISTER, not a timer: QA holds the
// destinations of the cartons between the scanner and blade A, QB those between A and B. A
// carton arriving at a blade pops the queue; one that is not for that blade is pushed onto the
// next one's. Timing the belt instead would mean a jam, a hand taking a carton off the line, or a
// change of speed override silently sorting the wrong box - a queue moves only when a beam says
// a carton actually went past.
//
// Destinations: 0 = take-away A, 1 = take-away B, 2 = straight through (a no-read).

START_EDGE := PB_START AND NOT PB_START_LAST;
PB_START_LAST := PB_START;
IF PB_CSTOP THEN
	STOP_REQ := TRUE;
END_IF;
SEL_CHANGED := SEL_AUTO <> SEL_LAST;
SEL_LAST := SEL_AUTO;

ESTOP := PB_ESTOP;
MASTER_EDGE := PB_MASTER AND NOT PB_MASTER_LAST;
PB_MASTER_LAST := PB_MASTER;
HOME_EDGE := PB_HOME AND NOT PB_HOME_LAST;
PB_HOME_LAST := PB_HOME;
IF ESTOP THEN
	MASTER_ON := FALSE;
	HOMED := FALSE;
ELSIF MASTER_EDGE THEN
	MASTER_ON := TRUE;
END_IF;
READY := MASTER_ON AND NOT ESTOP;

SCAN_EDGE := PE_IN AND NOT PE_IN_LAST;
UP_A_EDGE := PE_UP_A AND NOT PE_UP_A_LAST;
UP_B_EDGE := PE_UP_B AND NOT PE_UP_B_LAST;

CASE ST1_STEP OF
	0:	// idle
		DVA_EXEC := FALSE;
		DVB_EXEC := FALSE;
		CV_RUN := FALSE;
		SPA_RUN := FALSE;
		SPB_RUN := FALSE;
		EM_EN := FALSE;
		QA_H := 0;
		QA_T := 0;
		QA_N := 0;
		QB_H := 0;
		QB_T := 0;
		QB_N := 0;
		NEXT_DEST := 0;
		IF START_EDGE AND SEL_AUTO AND READY AND HOMED THEN
			STOP_REQ := FALSE;
			ST2_STEP := 100;
			ST3_STEP := 100;
			ST1_STEP := 10;
		END_IF;
	10:	// the line runs and the scanner reads every carton that goes by
		CV_RUN := TRUE;
		SPA_RUN := TRUE;
		SPB_RUN := TRUE;
		EM_EN := TRUE;
		IF SCAN_EDGE THEN
			IF QA_N >= 16 THEN
				ST1_STEP := 900;
			ELSE
				QA[QA_T] := NEXT_DEST;
				QA_T := (QA_T + 1) MOD 16;
				QA_N := QA_N + 1;
				NEXT_DEST := (NEXT_DEST + 1) MOD 3;
				CYCLE_CNT := CYCLE_CNT + 1;
			END_IF;
		END_IF;
		IF STOP_REQ AND QA_N = 0 AND QB_N = 0 THEN
			EM_EN := FALSE;
			ST1_STEP := 0;
		END_IF;
	800:	// HOME: the blades parked along the line, out of the path
		CV_RUN := FALSE;
		SPA_RUN := FALSE;
		SPB_RUN := FALSE;
		EM_EN := FALSE;
		DVA_TGT := 0.0;
		DVB_TGT := 0.0;
		DVA_EXEC := TRUE;
		DVB_EXEC := TRUE;
		IF DVA_DONE AND DVB_DONE THEN
			DVA_EXEC := FALSE;
			DVB_EXEC := FALSE;
			HOMED := TRUE;
			ST1_STEP := 0;
		END_IF;
	900:	// stuck, a runaway queue, or the selector was turned while running
		DVA_EXEC := FALSE;
		DVB_EXEC := FALSE;
		CV_RUN := FALSE;
		SPA_RUN := FALSE;
		SPB_RUN := FALSE;
		EM_EN := FALSE;
		IF START_EDGE AND SEL_AUTO THEN
			STOP_REQ := FALSE;
			ST1_STEP := 0;
		END_IF;
	910:	// the master circuit is open
		DVA_EXEC := FALSE;
		DVB_EXEC := FALSE;
		CV_RUN := FALSE;
		SPA_RUN := FALSE;
		SPB_RUN := FALSE;
		EM_EN := FALSE;
		IF READY THEN
			ST1_STEP := 0;
		END_IF;
END_CASE;

PE_IN_LAST := PE_IN;
RUNNING := ST1_STEP = 10;

// ---------------------------------------------------------- ST2: diverter A
IF NOT RUNNING THEN
	ST2_STEP := 0;
ELSE
	CASE ST2_STEP OF
		100:	// waiting for a carton; the queue says what this one is for
			IF UP_A_EDGE THEN
				IF QA_N > 0 THEN
					DEST := QA[QA_H];
					QA_H := (QA_H + 1) MOD 16;
					QA_N := QA_N - 1;
				ELSE
					DEST := 2;
				END_IF;
				IF DEST = 0 THEN
					ST2_STEP := 110;
				ELSE
					IF QB_N < 16 THEN
						QB[QB_T] := DEST;
						QB_T := (QB_T + 1) MOD 16;
						QB_N := QB_N + 1;
					END_IF;
					ST2_STEP := 130;
				END_IF;
			END_IF;
		110:	// the blade out, across the belt
			DVA_TGT := -45.0;
			DVA_EXEC := TRUE;
			IF DVA_DONE THEN
				ST2_STEP := 111;
			END_IF;
		111:
			DVA_EXEC := FALSE;
			IF NOT DVA_DONE THEN
				ST2_STEP := 112;
			END_IF;
		112:	// the carton rides the blade; the take-away beam says it arrived
			IF PE_A THEN
				ST2_STEP := 113;
			ELSIF T_DIV_A.Q THEN
				ST2_STEP := 900;
			END_IF;
		113:	// and it is CLEAR when that beam lets go again
			IF NOT PE_A THEN
				ST2_STEP := 120;
			END_IF;
		120:
			DVA_TGT := 0.0;
			DVA_EXEC := TRUE;
			IF DVA_DONE THEN
				ST2_STEP := 121;
			END_IF;
		121:
			DVA_EXEC := FALSE;
			IF NOT DVA_DONE THEN
				ST2_STEP := 100;
			END_IF;
		130:	// not for A: let it run on to B
			IF NOT PE_UP_A THEN
				ST2_STEP := 100;
			END_IF;
	ELSE
		ST2_STEP := 100;
	END_CASE;
END_IF;

// ---------------------------------------------------------- ST3: diverter B
IF NOT RUNNING THEN
	ST3_STEP := 0;
ELSE
	CASE ST3_STEP OF
		100:
			IF UP_B_EDGE THEN
				IF QB_N > 0 THEN
					DEST := QB[QB_H];
					QB_H := (QB_H + 1) MOD 16;
					QB_N := QB_N - 1;
				ELSE
					DEST := 2;
				END_IF;
				IF DEST = 1 THEN
					ST3_STEP := 110;
				ELSE
					ST3_STEP := 130;
				END_IF;
			END_IF;
		110:
			DVB_TGT := 45.0;
			DVB_EXEC := TRUE;
			IF DVB_DONE THEN
				ST3_STEP := 111;
			END_IF;
		111:
			DVB_EXEC := FALSE;
			IF NOT DVB_DONE THEN
				ST3_STEP := 112;
			END_IF;
		112:
			IF PE_B THEN
				ST3_STEP := 113;
			ELSIF T_DIV_B.Q THEN
				ST3_STEP := 900;
			END_IF;
		113:
			IF NOT PE_B THEN
				ST3_STEP := 120;
			END_IF;
		120:
			DVB_TGT := 0.0;
			DVB_EXEC := TRUE;
			IF DVB_DONE THEN
				ST3_STEP := 121;
			END_IF;
		121:
			DVB_EXEC := FALSE;
			IF NOT DVB_DONE THEN
				ST3_STEP := 100;
			END_IF;
		130:
			IF NOT PE_UP_B THEN
				ST3_STEP := 100;
			END_IF;
	ELSE
		ST3_STEP := 100;
	END_CASE;
END_IF;

PE_UP_A_LAST := PE_UP_A;
PE_UP_B_LAST := PE_UP_B;

// TONs after the CASE: their Q is read by the NEXT scan. A blade that is out and never sees its
// carton reach the take-away has lost it: that is a fault, not patience.
T_DIV_A(In := ST2_STEP = 112, PT := T#6s);
T_DIV_B(In := ST3_STEP = 112, PT := T#6s);

// A diverter step that stops moving is a jam. Its waiting step (100) is not: on a quiet line the
// next carton is as far away as the feed rate says. The TONs are called before the LAST copies
// are updated, so a step change gives them one scan of In = FALSE and resets them.
T_WD2(In := RUNNING AND ST2_STEP <> 100 AND ST2_STEP = STEP2_LAST, PT := T#20s);
T_WD3(In := RUNNING AND ST3_STEP <> 100 AND ST3_STEP = STEP3_LAST, PT := T#20s);
STEP2_LAST := ST2_STEP;
STEP3_LAST := ST3_STEP;
IF T_WD2.Q OR T_WD3.Q OR ST2_STEP = 900 OR ST3_STEP = 900 OR (SEL_CHANGED AND RUNNING) THEN
	ST1_STEP := 900;
	DVA_EXEC := FALSE;
	DVB_EXEC := FALSE;
	CV_RUN := FALSE;
	SPA_RUN := FALSE;
	SPB_RUN := FALSE;
	EM_EN := FALSE;
END_IF;

IF ESTOP THEN
	IF ST1_STEP <> 910 THEN
		ST1_STEP := 910;
	END_IF;
	DVA_EXEC := FALSE;
	DVB_EXEC := FALSE;
	CV_RUN := FALSE;
	SPA_RUN := FALSE;
	SPB_RUN := FALSE;
	EM_EN := FALSE;
ELSIF HOME_EDGE AND READY AND ST1_STEP = 0 THEN
	ST1_STEP := 800;
END_IF;

AUTO_RUN := ST1_STEP <> 0 AND ST1_STEP <> 800 AND ST1_STEP <> 900 AND ST1_STEP <> 910;
IND_ACTIVE := NOT SEL_AUTO AND NOT AUTO_RUN AND READY AND ST1_STEP <> 800;
IF IND_ACTIVE THEN
	IF IND_CV AND NOT IND_CV_LAST THEN
		MEM_CV := NOT MEM_CV;
	END_IF;
	IF IND_FEED AND NOT IND_FEED_LAST THEN
		MEM_FEED := NOT MEM_FEED;
	END_IF;
	IF IND_SPA AND NOT IND_SPA_LAST THEN
		MEM_SPA := NOT MEM_SPA;
	END_IF;
	IF IND_SPB AND NOT IND_SPB_LAST THEN
		MEM_SPB := NOT MEM_SPB;
	END_IF;
	CV_RUN := MEM_CV;
	EM_EN := MEM_FEED;
	SPA_RUN := MEM_SPA;
	SPB_RUN := MEM_SPB;
ELSE
	MEM_CV := FALSE;
	MEM_FEED := FALSE;
	MEM_SPA := FALSE;
	MEM_SPB := FALSE;
END_IF;
IND_CV_LAST := IND_CV;
IND_FEED_LAST := IND_FEED;
IND_SPA_LAST := IND_SPA;
IND_SPB_LAST := IND_SPB;
DVA_JOG_P := IND_ACTIVE AND IND_DVA_P;
DVA_JOG_N := IND_ACTIVE AND IND_DVA_N;
DVB_JOG_P := IND_ACTIVE AND IND_DVB_P;
DVB_JOG_N := IND_ACTIVE AND IND_DVB_N;

OVR := OVR_SET;
PL_START := AUTO_RUN;
PL_MASTER := MASTER_ON;
PL_HOME := HOMED;

(* ---- ce-insert.st ---- *)
VAR
	START_EDGE : BOOL;
	PB_START_LAST : BOOL;
	STOP_REQ : BOOL;
	SEL_LAST : BOOL := TRUE;
	SEL_CHANGED : BOOL;
	ESTOP : BOOL;
	READY : BOOL;
	MASTER_ON : BOOL;
	HOMED : BOOL;
	MASTER_EDGE : BOOL;
	PB_MASTER_LAST : BOOL;
	HOME_EDGE : BOOL;
	PB_HOME_LAST : BOOL;
	RUNNING : BOOL;
	TYPE1 : BOOL;
	A : INT;
	B : INT;
	I : INT;
	N : INT;
	SV_CENTER : LREAL;
	SV_LEFT : LREAL;
	SV_RIGHT : LREAL;
	SV_TGT : LREAL;
	HALF : INT;
	CHK : ARRAY[0..3] OF BOOL := [TRUE, TRUE, TRUE, TRUE];
	DIV_F : ARRAY[0..1] OF BOOL := [TRUE, TRUE];
	STP_DN : BOOL := TRUE;
	SEP_F : BOOL;
	PSH_F : BOOL;
	FDR : ARRAY[0..1] OF BOOL;
	MEM : ARRAY[0..3] OF BOOL;
	DELIV : BOOL;
	FLW : ARRAY[0..3] OF BOOL;
	SEEN1 : BOOL;
	SEEN2 : BOOL;
	FULL_IN : ARRAY[0..3] OF BOOL;
	FULL : ARRAY[0..3] OF BOOL;
	AS_CHK : ARRAY[0..3] OF BOOL;
	AS_UCHK : ARRAY[0..3] OF BOOL;
	FLW_IN : ARRAY[0..3] OF BOOL;
	T_FULL : ARRAY[0..3] OF TON;
	T_ST1OFF : TON;
	T_ST2OFF : TON;
	T_ST3FULL : TON;
	T_EXS : TON;
	T_DROP : TON;
	ST1_OFF : BOOL;
	ST2_OFF : BOOL;
	ST3_FULL : BOOL;
	EXS : BOOL;
	DROP_OFF : BOOL;
	ST2_READY : BOOL;
	T_WD1 : TON;
	T_WD2 : TON;
	T_WD3 : TON;
	STEP1_LAST : UDINT;
	STEP2_LAST : UDINT;
	STEP3_LAST : UDINT;
	JAM : BOOL;
	OUT_ON : BOOL;
	INDIVIDUAL : BOOL;
	IND_MOVE : BOOL;
	IND_TGT : LREAL;
	IND_C_LAST : BOOL;
	IND_L_LAST : BOOL;
	IND_R_LAST : BOOL;
	MEM_STP2 : BOOL;
	IND_STP2_LAST : BOOL;
	MEM_STP3 : BOOL;
	IND_STP3_LAST : BOOL;
	MEM_STP4 : BOOL;
	IND_STP4_LAST : BOOL;
	MEM_STP5 : BOOL;
	IND_STP5_LAST : BOOL;
	MEM_DIVL : BOOL;
	IND_DIVL_LAST : BOOL;
	MEM_DIVR : BOOL;
	IND_DIVR_LAST : BOOL;
	MEM_STP1 : BOOL;
	IND_STP1_LAST : BOOL;
	MEM_SEP : BOOL;
	IND_SEP_LAST : BOOL;
	MEM_PSH : BOOL;
	IND_PSH_LAST : BOOL;
	MEM_FDR1 : BOOL;
	IND_FDR1_LAST : BOOL;
	MEM_FDR2 : BOOL;
	IND_FDR2_LAST : BOOL;
END_VAR
// ce-insert: Denny's CE INSERT machine for spark plugs (tools/gen_ce_insert.js has the machine),
// ported from his NX1P2 program "Ce Insert Track". The same sequence runs without a PLC in
// ce-insert.ctl.js - keep the two in step.
//
// Three stations run at once and meet on shared state, as his Prg010/011/012 meet on GB010/011/012:
//   ST1  the running type's two gripper-stoppers open and pins run down to the divider until each
//        lane's FULL beam holds (then that gripper chucks); when the shuttle waits at a receiving
//        position the divider opens, the batch runs off, and it shuts once INSERT FLOW OUT has been
//        dark for 500 ms - after it has SEEN the batch go past.
//   ST2  the shuttle takes two batches on its four lanes: type 1 (left feeder, lanes 1-2) fills
//        shuttle lanes 1-2 at CENTER and 3-4 at LEFT; type 2 fills 3-4 at CENTER and 1-2 at RIGHT.
//        Full, it goes to CENTER and lifts STOPPER-1 onto the chute, while the chute is not full.
//   ST3  four pins at the chute end (SHUTTER EXIST 1-4): the separator takes them out of the queue,
//        goes back, the pusher pushes them over the receivers and they drop down the pipes.
//
// Not copied from his program, both found while porting: its ST3 drives the EJECTOR valve from the
// PUSHER symbols and the other way round (Denny confirmed the swap), and its ST2 Memory rung sets
// "shutter 3, 4 full" at POS4 with no batch delivered.

// BEGIN GENERATED - tools/gen_ce_insert.js
SV_CENTER := 110.0;
SV_LEFT := 30.0;
SV_RIGHT := 190.0;
// END GENERATED

START_EDGE := PB_START AND NOT PB_START_LAST;
PB_START_LAST := PB_START;
IF PB_CSTOP THEN
	STOP_REQ := TRUE;
END_IF;
SEL_CHANGED := SEL_AUTO <> SEL_LAST;
SEL_LAST := SEL_AUTO;
ESTOP := PB_ESTOP;
MASTER_EDGE := PB_MASTER AND NOT PB_MASTER_LAST;
PB_MASTER_LAST := PB_MASTER;
HOME_EDGE := PB_HOME AND NOT PB_HOME_LAST;
PB_HOME_LAST := PB_HOME;
IF ESTOP THEN
	MASTER_ON := FALSE;
	HOMED := FALSE;
ELSIF MASTER_EDGE THEN
	MASTER_ON := TRUE;
END_IF;
READY := MASTER_ON AND NOT ESTOP;
TYPE1 := NOT SEL_TYPE2;
IF TYPE1 THEN
	A := 0;
ELSE
	A := 2;
END_IF;
B := A + 1;

// The beams, debounced the way his LT timers do it.
FULL_IN[0] := PH_ST1_SHT1_FULL;
FULL_IN[1] := PH_ST1_SHT2_FULL;
FULL_IN[2] := PH_ST1_SHT3_FULL;
FULL_IN[3] := PH_ST1_SHT4_FULL;
FOR I := 0 TO 3 DO
	T_FULL[I](In := FULL_IN[I], PT := T#300ms);
	FULL[I] := T_FULL[I].Q;
END_FOR;
AS_CHK[0] := AS_ST1_STP2_CHK;
AS_CHK[1] := AS_ST1_STP3_CHK;
AS_CHK[2] := AS_ST1_STP4_CHK;
AS_CHK[3] := AS_ST1_STP5_CHK;
AS_UCHK[0] := AS_ST1_STP2_UCHK;
AS_UCHK[1] := AS_ST1_STP3_UCHK;
AS_UCHK[2] := AS_ST1_STP4_UCHK;
AS_UCHK[3] := AS_ST1_STP5_UCHK;
FLW_IN[0] := PH_ST3_SHT1_FLW_OUT;
FLW_IN[1] := PH_ST3_SHT2_FLW_OUT;
FLW_IN[2] := PH_ST3_SHT3_FLW_OUT;
FLW_IN[3] := PH_ST3_SHT4_FLW_OUT;
T_ST1OFF(In := NOT PH_ST1_INS_FLW_OUT, PT := T#500ms);
ST1_OFF := T_ST1OFF.Q;
T_ST2OFF(In := NOT PH_ST2_INS_FLW_OUT, PT := T#500ms);
ST2_OFF := T_ST2OFF.Q;
T_ST3FULL(In := PH_ST3_SHT_FULL, PT := T#300ms);
ST3_FULL := T_ST3FULL.Q;
T_EXS(In := PH_ST3_SHT1_EXS AND PH_ST3_SHT2_EXS AND PH_ST3_SHT3_EXS AND PH_ST3_SHT4_EXS, PT := T#200ms);
EXS := T_EXS.Q;
T_DROP(In := NOT (PH_ST3_SHT1_FLW_OUT OR PH_ST3_SHT2_FLW_OUT OR PH_ST3_SHT3_FLW_OUT OR PH_ST3_SHT4_FLW_OUT), PT := T#100ms);
DROP_OFF := T_DROP.Q;
// ST2 stands at a receiving position waiting for a batch (his GB011_11 / 12).
ST2_READY := ST2_STEP = 120;

// ---------------------------------------------------------------- ST1: supply feeder
CASE ST1_STEP OF
	0:	// idle
		FDR[0] := FALSE;
		FDR[1] := FALSE;
		IF START_EDGE AND SEL_AUTO AND READY AND HOMED AND AS_ST2_STP1_DN AND AS_ST3_EJC_BWD AND AS_ST3_PSH_BWD THEN
			STOP_REQ := FALSE;
			ST2_STEP := 100;
			ST3_STEP := 200;
			ST1_STEP := 10;
		END_IF;
	10:	// the running type's bowl feeds all the time; buffer, or discharge into a waiting shuttle
		FDR[0] := TYPE1;
		FDR[1] := NOT TYPE1;
		IF NOT (FULL[A] AND FULL[B]) THEN
			ST1_STEP := 20;
		ELSIF ST2_READY THEN
			ST1_STEP := 40;
		END_IF;
	20:	// buffering: both grippers of the pair open
		CHK[A] := FALSE;
		CHK[B] := FALSE;
		IF AS_UCHK[A] AND AS_UCHK[B] THEN
			ST1_STEP := 30;
		END_IF;
	30:	// each gripper chucks as soon as its own lane is full
		IF FULL[A] THEN
			CHK[A] := TRUE;
		END_IF;
		IF FULL[B] THEN
			CHK[B] := TRUE;
		END_IF;
		IF CHK[A] AND CHK[B] AND AS_CHK[A] AND AS_CHK[B] THEN
			ST1_STEP := 10;
		END_IF;
	40:	// discharging: the pair's divider opens
		IF TYPE1 THEN
			DIV_F[0] := FALSE;
		ELSE
			DIV_F[1] := FALSE;
		END_IF;
		SEEN1 := FALSE;
		IF (TYPE1 AND AS_ST1_LFT_DIV_BWD) OR (NOT TYPE1 AND AS_ST1_RGT_DIV_BWD) THEN
			ST1_STEP := 45;
		END_IF;
	45:	// the batch must be SEEN going past before "dark" means it has gone
		IF PH_ST1_INS_FLW_OUT THEN
			SEEN1 := TRUE;
		END_IF;
		IF SEEN1 AND ST1_OFF THEN
			ST1_STEP := 50;
		END_IF;
	50:
		DIV_F[0] := TRUE;
		DIV_F[1] := TRUE;
		IF AS_ST1_LFT_DIV_FWD AND AS_ST1_RGT_DIV_FWD THEN
			DELIV := TRUE;
			IF STOP_REQ THEN
				ST1_STEP := 0;
			ELSE
				ST1_STEP := 10;
			END_IF;
		END_IF;
	800:	// HOME: grippers chucked, dividers and STOPPER-1 closed, separator and pusher back, shuttle CENTER
		FOR I := 0 TO 3 DO
			CHK[I] := TRUE;
		END_FOR;
		DIV_F[0] := TRUE;
		DIV_F[1] := TRUE;
		STP_DN := TRUE;
		SEP_F := FALSE;
		PSH_F := FALSE;
		FDR[0] := FALSE;
		FDR[1] := FALSE;
		SV_ST2_TGT := SV_CENTER;
		SV_ST2_EXEC := TRUE;
		IF SV_ST2_DONE AND AS_ST1_STP2_CHK AND AS_ST1_STP3_CHK AND AS_ST1_STP4_CHK AND AS_ST1_STP5_CHK
				AND AS_ST1_LFT_DIV_FWD AND AS_ST1_RGT_DIV_FWD AND AS_ST2_STP1_DN AND AS_ST3_EJC_BWD AND AS_ST3_PSH_BWD THEN
			SV_ST2_EXEC := FALSE;
			FOR I := 0 TO 3 DO
				MEM[I] := FALSE;
			END_FOR;
			DELIV := FALSE;
			HOMED := TRUE;
			ST1_STEP := 0;
		END_IF;
	910:	// E-STOP
		FDR[0] := FALSE;
		FDR[1] := FALSE;
		SV_ST2_EXEC := FALSE;
		IF READY THEN
			ST1_STEP := 0;
		END_IF;
	900:	// FAULT: START acknowledges
		FDR[0] := FALSE;
		FDR[1] := FALSE;
		SV_ST2_EXEC := FALSE;
		IF START_EDGE AND SEL_AUTO THEN
			STOP_REQ := FALSE;
			ST1_STEP := 0;
		END_IF;
END_CASE;
RUNNING := (ST1_STEP <> 0) AND (ST1_STEP <> 800) AND (ST1_STEP <> 900) AND (ST1_STEP <> 910);

// ---------------------------------------------------------------- ST2: the shuttle
IF NOT RUNNING THEN
	ST2_STEP := 0;
ELSE
	CASE ST2_STEP OF
		100:	// decide
			N := 0;
			FOR I := 0 TO 3 DO
				IF MEM[I] THEN
					N := N + 1;
				END_IF;
			END_FOR;
			IF N = 4 THEN
				IF NOT ST3_FULL AND ST2_OFF THEN
					SV_TGT := SV_CENTER;
					ST2_STEP := 160;
				END_IF;
			ELSIF N = 0 THEN
				SV_TGT := SV_CENTER;
				IF TYPE1 THEN
					HALF := 0;
				ELSE
					HALF := 2;
				END_IF;
				ST2_STEP := 110;
			ELSIF TYPE1 AND MEM[0] AND MEM[1] AND NOT MEM[2] AND NOT MEM[3] THEN
				SV_TGT := SV_LEFT;
				HALF := 2;
				ST2_STEP := 110;
			ELSIF NOT TYPE1 AND MEM[2] AND MEM[3] AND NOT MEM[0] AND NOT MEM[1] THEN
				SV_TGT := SV_RIGHT;
				HALF := 0;
				ST2_STEP := 110;
			ELSIF NOT ST3_FULL AND ST2_OFF THEN
				// half a load of the other type (the type was changed): run it off
				SV_TGT := SV_CENTER;
				ST2_STEP := 160;
			END_IF;
		110:	// Execute is a LEVEL held until Done
			SV_ST2_TGT := SV_TGT;
			SV_ST2_EXEC := TRUE;
			IF SV_ST2_DONE THEN
				SV_ST2_EXEC := FALSE;
				ST2_STEP := 115;
			END_IF;
		115:
			IF NOT SV_ST2_DONE THEN
				ST2_STEP := 120;
			END_IF;
		120:	// at a receiving position: ST1 discharges into the lanes in front of it
			IF DELIV THEN
				DELIV := FALSE;
				MEM[HALF] := TRUE;
				MEM[HALF + 1] := TRUE;
				ST2_STEP := 100;
			END_IF;
		160:
			SV_ST2_TGT := SV_CENTER;
			SV_ST2_EXEC := TRUE;
			IF SV_ST2_DONE THEN
				SV_ST2_EXEC := FALSE;
				ST2_STEP := 165;
			END_IF;
		165:
			IF NOT SV_ST2_DONE THEN
				ST2_STEP := 170;
			END_IF;
		170:	// STOPPER-1 up: all four lanes run onto the chute
			STP_DN := FALSE;
			SEEN2 := FALSE;
			IF AS_ST2_STP1_UP THEN
				ST2_STEP := 175;
			END_IF;
		175:
			IF PH_ST2_INS_FLW_OUT THEN
				SEEN2 := TRUE;
			END_IF;
			IF SEEN2 AND ST2_OFF THEN
				ST2_STEP := 180;
			END_IF;
		180:
			STP_DN := TRUE;
			IF AS_ST2_STP1_DN THEN
				FOR I := 0 TO 3 DO
					MEM[I] := FALSE;
				END_FOR;
				ST2_STEP := 100;
			END_IF;
		ELSE
			ST2_STEP := 100;
	END_CASE;
END_IF;

// ---------------------------------------------------------------- ST3: CE eject
IF NOT RUNNING THEN
	ST3_STEP := 0;
ELSE
	CASE ST3_STEP OF
		200:	// four pins at the chute end
			SEP_F := FALSE;
			PSH_F := FALSE;
			IF EXS THEN
				ST3_STEP := 210;
			END_IF;
		210:	// the separator takes them out of the queue
			SEP_F := TRUE;
			IF AS_ST3_EJC_FWD THEN
				ST3_STEP := 215;
			END_IF;
		215:	// still in the beams, in the slots
			IF PH_ST3_SHT1_EXS AND PH_ST3_SHT2_EXS AND PH_ST3_SHT3_EXS AND PH_ST3_SHT4_EXS THEN
				ST3_STEP := 220;
			END_IF;
		220:
			SEP_F := FALSE;
			IF AS_ST3_EJC_BWD THEN
				FOR I := 0 TO 3 DO
					FLW[I] := FALSE;
				END_FOR;
				ST3_STEP := 230;
			END_IF;
		230:	// the pusher takes them over the receivers: they drop
			PSH_F := TRUE;
			IF AS_ST3_PSH_FWD THEN
				ST3_STEP := 240;
			END_IF;
		240:
			PSH_F := FALSE;
			IF AS_ST3_PSH_BWD THEN
				ST3_STEP := 250;
			END_IF;
		250:	// every pin went down its pipe, and none is still in a beam
			IF FLW[0] AND FLW[1] AND FLW[2] AND FLW[3] AND DROP_OFF THEN
				CYCLE_CNT := CYCLE_CNT + 1;
				ST3_STEP := 200;
			END_IF;
		ELSE
			ST3_STEP := 200;
	END_CASE;
END_IF;
IF (ST3_STEP >= 230) AND (ST3_STEP <= 250) THEN
	FOR I := 0 TO 3 DO
		IF FLW_IN[I] THEN
			FLW[I] := TRUE;
		END_IF;
	END_FOR;
END_IF;

// Watchdog, one per station, on the steps that MOVE something (waits for material excluded).
T_WD1(In := (ST1_STEP = STEP1_LAST) AND RUNNING AND (ST1_STEP <> 10), PT := T#15s);
T_WD2(In := (ST2_STEP = STEP2_LAST) AND RUNNING AND (ST2_STEP <> 100) AND (ST2_STEP <> 120), PT := T#15s);
T_WD3(In := (ST3_STEP = STEP3_LAST) AND RUNNING AND (ST3_STEP <> 200), PT := T#15s);
IF ST1_STEP <> STEP1_LAST THEN
	STEP1_LAST := ST1_STEP;
END_IF;
IF ST2_STEP <> STEP2_LAST THEN
	STEP2_LAST := ST2_STEP;
END_IF;
IF ST3_STEP <> STEP3_LAST THEN
	STEP3_LAST := ST3_STEP;
END_IF;
JAM := T_WD1.Q OR T_WD2.Q OR T_WD3.Q;
IF RUNNING AND (JAM OR SEL_CHANGED) THEN
	ST1_STEP := 900;
	ST2_STEP := 0;
	ST3_STEP := 0;
	SV_ST2_EXEC := FALSE;
	FDR[0] := FALSE;
	FDR[1] := FALSE;
END_IF;
IF ESTOP THEN
	IF ST1_STEP <> 910 THEN
		ST1_STEP := 910;
	END_IF;
	ST2_STEP := 0;
	ST3_STEP := 0;
	SV_ST2_EXEC := FALSE;
	FDR[0] := FALSE;
	FDR[1] := FALSE;
ELSIF HOME_EDGE AND READY AND (ST1_STEP = 0) THEN
	ST1_STEP := 800;
END_IF;

AUTO_RUN := (ST1_STEP <> 0) AND (ST1_STEP <> 800) AND (ST1_STEP <> 900) AND (ST1_STEP <> 910);

// Individual operation: momentary buttons, a PLC toggle memory per actuator, cleared when
// INDIVIDUAL ends. The shuttle position buttons start one move each; Execute drops at Done.
INDIVIDUAL := NOT SEL_AUTO AND NOT AUTO_RUN AND READY AND (ST1_STEP <> 800);
IF INDIVIDUAL THEN
	IF IND_STP2 AND NOT IND_STP2_LAST THEN
		MEM_STP2 := NOT MEM_STP2;
	END_IF;
	IF IND_STP3 AND NOT IND_STP3_LAST THEN
		MEM_STP3 := NOT MEM_STP3;
	END_IF;
	IF IND_STP4 AND NOT IND_STP4_LAST THEN
		MEM_STP4 := NOT MEM_STP4;
	END_IF;
	IF IND_STP5 AND NOT IND_STP5_LAST THEN
		MEM_STP5 := NOT MEM_STP5;
	END_IF;
	IF IND_DIVL AND NOT IND_DIVL_LAST THEN
		MEM_DIVL := NOT MEM_DIVL;
	END_IF;
	IF IND_DIVR AND NOT IND_DIVR_LAST THEN
		MEM_DIVR := NOT MEM_DIVR;
	END_IF;
	IF IND_STP1 AND NOT IND_STP1_LAST THEN
		MEM_STP1 := NOT MEM_STP1;
	END_IF;
	IF IND_SEP AND NOT IND_SEP_LAST THEN
		MEM_SEP := NOT MEM_SEP;
	END_IF;
	IF IND_PSH AND NOT IND_PSH_LAST THEN
		MEM_PSH := NOT MEM_PSH;
	END_IF;
	IF IND_FDR1 AND NOT IND_FDR1_LAST THEN
		MEM_FDR1 := NOT MEM_FDR1;
	END_IF;
	IF IND_FDR2 AND NOT IND_FDR2_LAST THEN
		MEM_FDR2 := NOT MEM_FDR2;
	END_IF;
	CHK[0] := NOT MEM_STP2;
	CHK[1] := NOT MEM_STP3;
	CHK[2] := NOT MEM_STP4;
	CHK[3] := NOT MEM_STP5;
	DIV_F[0] := NOT MEM_DIVL;
	DIV_F[1] := NOT MEM_DIVR;
	STP_DN := NOT MEM_STP1;
	SEP_F := MEM_SEP;
	PSH_F := MEM_PSH;
	FDR[0] := MEM_FDR1;
	FDR[1] := MEM_FDR2;
	IF NOT IND_MOVE AND ((IND_SV_CTR AND NOT IND_C_LAST) OR (IND_SV_LFT AND NOT IND_L_LAST) OR (IND_SV_RGT AND NOT IND_R_LAST)) THEN
		IND_MOVE := TRUE;
		IF IND_SV_CTR THEN
			IND_TGT := SV_CENTER;
		ELSIF IND_SV_LFT THEN
			IND_TGT := SV_LEFT;
		ELSE
			IND_TGT := SV_RIGHT;
		END_IF;
	END_IF;
	IND_C_LAST := IND_SV_CTR;
	IND_L_LAST := IND_SV_LFT;
	IND_R_LAST := IND_SV_RGT;
	SV_ST2_TGT := IND_TGT;
	SV_ST2_EXEC := IND_MOVE;
	IF IND_MOVE AND SV_ST2_DONE THEN
		IND_MOVE := FALSE;
	END_IF;
ELSE
	MEM_STP2 := FALSE;
	MEM_STP3 := FALSE;
	MEM_STP4 := FALSE;
	MEM_STP5 := FALSE;
	MEM_DIVL := FALSE;
	MEM_DIVR := FALSE;
	MEM_STP1 := FALSE;
	MEM_SEP := FALSE;
	MEM_PSH := FALSE;
	MEM_FDR1 := FALSE;
	MEM_FDR2 := FALSE;
	IND_MOVE := FALSE;
	IND_C_LAST := FALSE;
	IND_L_LAST := FALSE;
	IND_R_LAST := FALSE;
END_IF;
IND_STP2_LAST := IND_STP2;
IND_STP3_LAST := IND_STP3;
IND_STP4_LAST := IND_STP4;
IND_STP5_LAST := IND_STP5;
IND_DIVL_LAST := IND_DIVL;
IND_DIVR_LAST := IND_DIVR;
IND_STP1_LAST := IND_STP1;
IND_SEP_LAST := IND_SEP;
IND_PSH_LAST := IND_PSH;
IND_FDR1_LAST := IND_FDR1;
IND_FDR2_LAST := IND_FDR2;

// Solenoids from where each actuator is told to be. Without MASTER ON (and on E-STOP) the master
// circuit is open and every coil drops: a double-solenoid valve then holds where it is.
OUT_ON := READY;
SOL_ST1_STP2_CHK := OUT_ON AND CHK[0];
SOL_ST1_STP2_UCHK := OUT_ON AND NOT CHK[0];
SOL_ST1_STP3_CHK := OUT_ON AND CHK[1];
SOL_ST1_STP3_UCHK := OUT_ON AND NOT CHK[1];
SOL_ST1_STP4_CHK := OUT_ON AND CHK[2];
SOL_ST1_STP4_UCHK := OUT_ON AND NOT CHK[2];
SOL_ST1_STP5_CHK := OUT_ON AND CHK[3];
SOL_ST1_STP5_UCHK := OUT_ON AND NOT CHK[3];
SOL_ST1_LFT_DIV_FWD := OUT_ON AND DIV_F[0];
SOL_ST1_LFT_DIV_BWD := OUT_ON AND NOT DIV_F[0];
SOL_ST1_RGT_DIV_FWD := OUT_ON AND DIV_F[1];
SOL_ST1_RGT_DIV_BWD := OUT_ON AND NOT DIV_F[1];
SOL_ST2_STP1_DN := OUT_ON AND STP_DN;
SOL_ST2_STP1_UP := OUT_ON AND NOT STP_DN;
SOL_ST3_EJC_FWD := OUT_ON AND SEP_F;
SOL_ST3_EJC_BWD := OUT_ON AND NOT SEP_F;
SOL_ST3_PSH_FWD := OUT_ON AND PSH_F;
SOL_ST3_PSH_BWD := OUT_ON AND NOT PSH_F;
CR_ST1_PART_FDR1_STR := OUT_ON AND FDR[0];
CR_ST1_PART_FDR2_STR := OUT_ON AND FDR[1];

OVR := OVR_SET;
SV_ST2_JOG_P := INDIVIDUAL AND IND_SV_P;
SV_ST2_JOG_N := INDIVIDUAL AND IND_SV_N;
PL_START := AUTO_RUN;
PL_MASTER := MASTER_ON;
PL_HOME := HOMED;
PL_SV_CTR := ABS(SV_ST2_POS - SV_CENTER) < 0.5;
PL_SV_LFT := ABS(SV_ST2_POS - SV_LEFT) < 0.5;
PL_SV_RGT := ABS(SV_ST2_POS - SV_RIGHT) < 0.5;

(* ---- cyl-on-slide.st ---- *)
VAR
	START_EDGE : BOOL;
	PB_START_LAST : BOOL;
	STOP_REQ : BOOL;
	T_DWELL : TON;
END_VAR
// cyl-on-slide: slide to the press position, press down, dwell, press up, slide home, repeat
// until STOP. The same sequence runs without a PLC in cyl-on-slide.ctl.js.
//
// The servo handshake is MC_MoveAbsolute's: Execute is a LEVEL held until Done, and Done must
// be seen to drop before the next Execute. The plant samples PLC outputs every ~16 ms, so a
// one-scan pulse would be missed.

START_EDGE := PB_START AND NOT PB_START_LAST;
PB_START_LAST := PB_START;
IF PB_STOP THEN
	STOP_REQ := TRUE;
END_IF;

CASE ST1_STEP OF
	0:	// idle at home, cylinder up
		SOL_ST1_PRSS_CYL_DN := FALSE;
		SOL_ST1_PRSS_CYL_UP := TRUE;
		SV1_EXEC := FALSE;
		IF START_EDGE AND AS_ST1_PRSS_CYL_UP AND SV1_INPOS AND NOT SV1_DONE THEN
			STOP_REQ := FALSE;
			ST1_STEP := 10;
		END_IF;
	10:	// slide to the press position
		SV1_TGT := 400.0;
		SV1_EXEC := TRUE;
		IF SV1_DONE THEN
			SV1_EXEC := FALSE;
			ST1_STEP := 20;
		END_IF;
	20:	// wait until the plant has seen Execute drop
		IF NOT SV1_DONE THEN
			ST1_STEP := 30;
		END_IF;
	30:	// press down
		SOL_ST1_PRSS_CYL_UP := FALSE;
		SOL_ST1_PRSS_CYL_DN := TRUE;
		IF AS_ST1_PRSS_CYL_DN THEN
			ST1_STEP := 40;
		END_IF;
	40:	// dwell on the part
		IF T_DWELL.Q THEN
			ST1_STEP := 50;
		END_IF;
	50:	// press up
		SOL_ST1_PRSS_CYL_DN := FALSE;
		SOL_ST1_PRSS_CYL_UP := TRUE;
		IF AS_ST1_PRSS_CYL_UP THEN
			ST1_STEP := 60;
		END_IF;
	60:	// slide home
		SV1_TGT := 0.0;
		SV1_EXEC := TRUE;
		IF SV1_DONE THEN
			SV1_EXEC := FALSE;
			ST1_STEP := 70;
		END_IF;
	70:	// cycle complete
		IF NOT SV1_DONE THEN
			CYCLE_CNT := CYCLE_CNT + 1;
			IF STOP_REQ THEN
				ST1_STEP := 0;
			ELSE
				ST1_STEP := 10;
			END_IF;
		END_IF;
END_CASE;

T_DWELL(In := (ST1_STEP = 40), PT := T#300ms);
AUTO_RUN := ST1_STEP <> 0;
PL_START := AUTO_RUN;

(* ---- gripper-transfer.st ---- *)
VAR
	START_EDGE : BOOL;
	PB_START_LAST : BOOL;
	STOP_REQ : BOOL;
	SEL_LAST : BOOL := TRUE;
	SEL_CHANGED : BOOL;
	EM_LAST : UDINT;
	T_SETTLE : TON;
	T_GRIP : TON;
	T_WD : TON;
	STEP_LAST : UDINT;
	GONE : UDINT;
	MEM_CV1 : BOOL;
	IND_CV1_LAST : BOOL;
	MEM_CV2 : BOOL;
	IND_CV2_LAST : BOOL;
	MEM_LIFT : BOOL;
	IND_LIFT_LAST : BOOL;
	MEM_TRAV : BOOL;
	IND_TRAV_LAST : BOOL;
	MEM_GRIP : BOOL;
	IND_GRIP_LAST : BOOL;
	ESTOP : BOOL;
	READY : BOOL;
	MASTER_ON : BOOL;
	HOMED : BOOL;
	MASTER_EDGE : BOOL;
	PB_MASTER_LAST : BOOL;
	HOME_EDGE : BOOL;
	PB_HOME_LAST : BOOL;
END_VAR
// gripper-transfer: a part rides the infeed belt to the pick beam and stops. A 2-finger gripper on
// a pneumatic lift on a pneumatic traverse picks it, carries it over the outfeed belt (running
// across, the other way) and sets it down. Repeat until STOP. The same sequence runs without a
// PLC in gripper-transfer.ctl.js.
//
// A gripper has no "part gripped" switch: after the closing time the fingers are either stopped
// by the part (neither switch on) or fully closed on nothing (CLOSED on). A missed grip is a
// FAULT, not a cycle with an empty gripper.
//
// Waiting steps wait for an INVARIANT, not for a counter to move: every part loaded has left.
//
// The panel has a selector AUTO / INDIVIDUAL: START only in AUTO, the individual buttons only in
// INDIVIDUAL, and a change while the sequence runs is a FAULT, not a pause.

START_EDGE := PB_START AND NOT PB_START_LAST;
PB_START_LAST := PB_START;
IF PB_CSTOP THEN
	STOP_REQ := TRUE;
END_IF;
SEL_CHANGED := SEL_AUTO <> SEL_LAST;
SEL_LAST := SEL_AUTO;

// The master circuit, as on the cell panel: E-STOP is a latching mushroom, MASTER ON energises
// the machine, and nothing runs without it. An E-STOP also loses the home position.
ESTOP := PB_ESTOP;
MASTER_EDGE := PB_MASTER AND NOT PB_MASTER_LAST;
PB_MASTER_LAST := PB_MASTER;
HOME_EDGE := PB_HOME AND NOT PB_HOME_LAST;
PB_HOME_LAST := PB_HOME;
IF ESTOP THEN
	MASTER_ON := FALSE;
	HOMED := FALSE;
ELSIF MASTER_EDGE THEN
	MASTER_ON := TRUE;
END_IF;
READY := MASTER_ON AND NOT ESTOP;

// A write-off goes STALE when the part turns up after all, and then RM + GONE runs PAST EM and
// the step waiting on that invariant stops waiting at all. GONE is a UDINT, so the subtraction
// underflows to about 4 billion when RM is ahead: guard before you subtract.
IF RM_CNT >= EM_CNT THEN
	GONE := 0;
ELSIF RM_CNT + GONE > EM_CNT THEN
	GONE := EM_CNT - RM_CNT;
END_IF;
CASE ST1_STEP OF
	0:	// idle: lift up, traverse in, gripper open
		CV1_RUN := FALSE;
		CV2_RUN := FALSE;
		EM_EMIT := FALSE;
		GRIP_CLOSE := FALSE;
		SOL_Z_DN := FALSE;
		SOL_Z_UP := TRUE;
		SOL_Y_OUT := FALSE;
		SOL_Y_IN := TRUE;
		IF START_EDGE AND SEL_AUTO AND READY AND HOMED AND AS_Z_UP AND AS_Y_IN AND GRIP_OPEN THEN
			STOP_REQ := FALSE;
			EM_LAST := EM_CNT;
			ST1_STEP := 10;
		END_IF;
	10:	// outfeed belt on, feed one part
		CV2_RUN := TRUE;
		EM_EMIT := TRUE;
		IF EM_CNT <> EM_LAST THEN
			EM_EMIT := FALSE;
			ST1_STEP := 15;
		END_IF;
	15:	// the pick beam must be clear before this part runs to it
		CV1_RUN := TRUE;
		IF NOT PE_PICK THEN
			ST1_STEP := 20;
		END_IF;
	20:	// carry it to the pick beam
		CV1_RUN := TRUE;
		IF PE_PICK THEN
			CV1_RUN := FALSE;
			ST1_STEP := 30;
		END_IF;
	30:	// let it settle under the gripper
		IF T_SETTLE.Q THEN
			ST1_STEP := 40;
		END_IF;
	40:	// lift down
		SOL_Z_UP := FALSE;
		SOL_Z_DN := TRUE;
		IF AS_Z_DN THEN
			ST1_STEP := 50;
		END_IF;
	50:	// close: stopped by the part = gripped, fully closed = missed
		GRIP_CLOSE := TRUE;
		IF T_GRIP.Q THEN
			IF GRIP_CLOSED THEN
				ST1_STEP := 900;
			ELSE
				ST1_STEP := 60;
			END_IF;
		END_IF;
	60:	// lift up with the part
		SOL_Z_DN := FALSE;
		SOL_Z_UP := TRUE;
		IF AS_Z_UP THEN
			ST1_STEP := 70;
		END_IF;
	70:	// traverse out over the outfeed belt
		SOL_Y_IN := FALSE;
		SOL_Y_OUT := TRUE;
		IF AS_Y_OUT THEN
			ST1_STEP := 80;
		END_IF;
	80:	// lift down onto the belt
		SOL_Z_UP := FALSE;
		SOL_Z_DN := TRUE;
		IF AS_Z_DN THEN
			ST1_STEP := 90;
		END_IF;
	90:	// open: the part is on the belt
		GRIP_CLOSE := FALSE;
		IF GRIP_OPEN THEN
			ST1_STEP := 100;
		END_IF;
	100:	// lift up
		SOL_Z_DN := FALSE;
		SOL_Z_UP := TRUE;
		IF AS_Z_UP THEN
			ST1_STEP := 110;
		END_IF;
	110:	// traverse in
		SOL_Y_OUT := FALSE;
		SOL_Y_IN := TRUE;
		IF AS_Y_IN THEN
			ST1_STEP := 120;
		END_IF;
	120:	// the outfeed belt carries the part away: everything loaded must have left
		IF RM_CNT + GONE >= EM_CNT THEN
			CYCLE_CNT := CYCLE_CNT + 1;
			IF STOP_REQ THEN
				ST1_STEP := 0;
			ELSE
				EM_LAST := EM_CNT;
				ST1_STEP := 10;
			END_IF;
		END_IF;
	800:	// HOME: lift up and traverse in. The gripper is left alone: a real machine does not drop the part it holds
		CV1_RUN := FALSE;
		CV2_RUN := FALSE;
		EM_EMIT := FALSE;
		SOL_Z_DN := FALSE;
		SOL_Z_UP := TRUE;
		SOL_Y_OUT := FALSE;
		SOL_Y_IN := TRUE;
		IF AS_Z_UP AND AS_Y_IN THEN
			HOMED := TRUE;
			ST1_STEP := 0;
		END_IF;
	910:	// E-STOP: the master circuit is open, so every solenoid de-energises - which is what
		// really happens: a 5/2 single-solenoid valve springs back, a double one holds. The holders keep their parts: a real machine does not let go when the power drops.
		CV1_RUN := FALSE;
		EM_EMIT := FALSE;
		SOL_Y_OUT := FALSE;
		SOL_Y_IN := FALSE;
		SOL_Z_DN := FALSE;
		SOL_Z_UP := FALSE;
		CV2_RUN := FALSE;
		IF READY THEN	// MASTER ON after the mushroom is released
			ST1_STEP := 0;
		END_IF;
	900:	// FAULT: a step stopped moving, the gripper closed on nothing, or the selector was turned
		// while running. Belts and feeding off; the gripper and the cylinders stay where they are.
		CV1_RUN := FALSE;
		CV2_RUN := FALSE;
		EM_EMIT := FALSE;
		IF START_EDGE AND SEL_AUTO THEN
			STOP_REQ := FALSE;
			// Acknowledging writes off whatever never reached the outfeed. Only HERE.
			GONE := EM_CNT - RM_CNT;
			ST1_STEP := 0;
		END_IF;
END_CASE;

T_SETTLE(In := (ST1_STEP = 30), PT := T#300ms);
T_GRIP(In := (ST1_STEP = 50), PT := T#400ms);

// Watchdog: a running step that stops moving is a jam, not patience. A selector change while
// running trips the same way.
T_WD(In := (ST1_STEP = STEP_LAST) AND (ST1_STEP <> 0) AND (ST1_STEP <> 900) AND (ST1_STEP <> 910), PT := T#15s);
IF ST1_STEP <> STEP_LAST THEN
	STEP_LAST := ST1_STEP;
END_IF;
IF T_WD.Q OR (SEL_CHANGED AND (ST1_STEP <> 0) AND (ST1_STEP <> 900) AND (ST1_STEP <> 910)) THEN
	ST1_STEP := 900;
	CV1_RUN := FALSE;
	CV2_RUN := FALSE;
	EM_EMIT := FALSE;
END_IF;

// E-STOP at any moment, and the HOME button when the machine is energised and idle.
IF ESTOP THEN
	IF ST1_STEP <> 910 THEN
		ST1_STEP := 910;
	END_IF;
	CV1_RUN := FALSE;
	EM_EMIT := FALSE;
	SOL_Y_OUT := FALSE;
	SOL_Y_IN := FALSE;
	SOL_Z_DN := FALSE;
	SOL_Z_UP := FALSE;
	CV2_RUN := FALSE;
ELSIF HOME_EDGE AND READY AND (ST1_STEP = 0) THEN
	ST1_STEP := 800;
END_IF;

AUTO_RUN := (ST1_STEP <> 0) AND (ST1_STEP <> 800) AND (ST1_STEP <> 900) AND (ST1_STEP <> 910);

// Individual operation: momentary buttons, a PLC toggle memory per actuator, cleared when INDIVIDUAL
// ends. The feed button pulses one part.
IF NOT SEL_AUTO AND NOT AUTO_RUN AND READY AND (ST1_STEP <> 800) THEN
	IF IND_CV1 AND NOT IND_CV1_LAST THEN
		MEM_CV1 := NOT MEM_CV1;
	END_IF;
	IF IND_CV2 AND NOT IND_CV2_LAST THEN
		MEM_CV2 := NOT MEM_CV2;
	END_IF;
	IF IND_LIFT AND NOT IND_LIFT_LAST THEN
		MEM_LIFT := NOT MEM_LIFT;
	END_IF;
	IF IND_TRAV AND NOT IND_TRAV_LAST THEN
		MEM_TRAV := NOT MEM_TRAV;
	END_IF;
	IF IND_GRIP AND NOT IND_GRIP_LAST THEN
		MEM_GRIP := NOT MEM_GRIP;
	END_IF;
	CV1_RUN := MEM_CV1;
	CV2_RUN := MEM_CV2;
	EM_EMIT := IND_FEED;
	SOL_Z_DN := MEM_LIFT;
	SOL_Z_UP := NOT MEM_LIFT;
	SOL_Y_OUT := MEM_TRAV;
	SOL_Y_IN := NOT MEM_TRAV;
	GRIP_CLOSE := MEM_GRIP;
ELSE
	MEM_CV1 := FALSE;
	MEM_CV2 := FALSE;
	MEM_LIFT := FALSE;
	MEM_TRAV := FALSE;
	MEM_GRIP := FALSE;
END_IF;
IND_CV1_LAST := IND_CV1;
IND_CV2_LAST := IND_CV2;
IND_LIFT_LAST := IND_LIFT;
IND_TRAV_LAST := IND_TRAV;
IND_GRIP_LAST := IND_GRIP;

// The speed override the operator dialled in, passed on to the axes and the belts.
OVR := OVR_SET;

PL_START := AUTO_RUN;
PL_MASTER := MASTER_ON;
PL_HOME := HOMED;

(* ---- lathe-line.st ---- *)
VAR
	START_EDGE : BOOL;
	PB_START_LAST : BOOL;
	STOP_REQ : BOOL;
	SEL_LAST : BOOL := TRUE;
	SEL_CHANGED : BOOL;
	T_WD : TON;
	T_GRIP : TON;
	T_SETTLE1 : TON;
	T_SETTLE2 : TON;
	T_DROP1 : TON;
	T_DROP2 : TON;
	T_CUT1 : TON;
	T_CUT2 : TON;
	T_WD4 : TON;
	T_WD5 : TON;
	STEP_LAST : UDINT;
	TGT : UINT;
	GO_POSE : UINT;
	GO_RAIL : UINT;
	HAS_RAW : BOOL;
	HAS_FIN : BOOL;
	M1_STATE : UINT;
	M2_STATE : UINT;
	S1_GO : BOOL;
	S2_GO : BOOL;
	ALL_DONE : BOOL;
	ALL_CLEAR : BOOL;
	COND : BOOL;
	MEM_A : BOOL;
	MEM_B : BOOL;
	MEM_D1 : BOOL;
	MEM_D2 : BOOL;
	MEM_L1 : BOOL;
	MEM_L2 : BOOL;
	IND_A_LAST : BOOL;
	IND_B_LAST : BOOL;
	IND_D1_LAST : BOOL;
	IND_D2_LAST : BOOL;
	IND_L1_LAST : BOOL;
	IND_L2_LAST : BOOL;
	IND_ACTIVE : BOOL;
	RUNNING : BOOL;
	ESTOP : BOOL;
	READY : BOOL;
	MASTER_ON : BOOL;
	HOMED : BOOL;
	MASTER_EDGE : BOOL;
	PB_MASTER_LAST : BOOL;
	HOME_EDGE : BOOL;
	PB_HOME_LAST : BOOL;
END_VAR
// lathe-line: a DENSO VS-087 hanging from a traverse beam serves two TAKISAWA TCC-2000 lathes
// (OP10 then OP20) standing side by side, fed by ONE conveyor along their fronts. At each machine
// a stopper pops up out of the belt and a pin lift raises the part to the robot; the same pin
// hands over the raw part and takes the finished one back. The same sequence runs without a PLC
// in lathe-line.ctl.js - keep the two in step.
//
// The hand is a 90 degree DOUBLE hand: A along the flange axis for raw parts, B across it for
// finished ones, so one door opening serves the whole exchange.
//
// A grip is confirmed by the OPEN switch DROPPING, never by CLOSED: CLOSED sits at full close, so
// with a part between the fingers it never comes on.
//
// The joint targets are set by the CASE GO_POSE block at the bottom, which is GENERATED from the
// same IK run as the controller's table (tools/gen_lathe_line.js): 66 angles typed into two
// programs by hand drift, and the drift is silent.

START_EDGE := PB_START AND NOT PB_START_LAST;
PB_START_LAST := PB_START;
IF PB_CSTOP THEN
	STOP_REQ := TRUE;
END_IF;
SEL_CHANGED := SEL_AUTO <> SEL_LAST;
SEL_LAST := SEL_AUTO;

ESTOP := PB_ESTOP;
MASTER_EDGE := PB_MASTER AND NOT PB_MASTER_LAST;
PB_MASTER_LAST := PB_MASTER;
HOME_EDGE := PB_HOME AND NOT PB_HOME_LAST;
PB_HOME_LAST := PB_HOME;
IF ESTOP THEN
	MASTER_ON := FALSE;
	HOMED := FALSE;
ELSIF MASTER_EDGE THEN
	MASTER_ON := TRUE;
END_IF;
READY := MASTER_ON AND NOT ESTOP;

ALL_DONE := J1_DONE AND J2_DONE AND J3_DONE AND J4_DONE AND J5_DONE AND J6_DONE;
ALL_CLEAR := NOT J1_DONE AND NOT J2_DONE AND NOT J3_DONE AND NOT J4_DONE AND NOT J5_DONE AND NOT J6_DONE;
GO_POSE := 0;

CASE ST1_STEP OF
	0:	// idle
		J1_EXEC := FALSE;
		J2_EXEC := FALSE;
		J3_EXEC := FALSE;
		J4_EXEC := FALSE;
		J5_EXEC := FALSE;
		J6_EXEC := FALSE;
		RX_EXEC := FALSE;
		EM_IN_EMIT := FALSE;
		CV_RUN := FALSE;
		GRIP_A := FALSE;
		GRIP_B := FALSE;
		SOL_M1_DOOR := FALSE;
		SOL_M2_DOOR := FALSE;
		M1_CHUCK := TRUE;
		M2_CHUCK := TRUE;
		HAS_RAW := FALSE;
		HAS_FIN := FALSE;
		IF START_EDGE AND SEL_AUTO AND READY AND HOMED THEN
			STOP_REQ := FALSE;
			ST2_STEP := 100;
			ST3_STEP := 100;
			ST4_STEP := 200;
			ST5_STEP := 200;
			ST1_STEP := 10;
		END_IF;
	10:	// which machine: one with a finished part first, it is holding one hostage
		HAS_RAW := FALSE;
		HAS_FIN := FALSE;
		// The pin must be UP with a raw part on it, every time: the robot gives the pin a finished
		// part back at the end of the visit, and what guarantees the pin is free then is that the
		// robot took what was on it. Going for a finished part with the pin empty cornered the
		// cell - the station cannot present an empty pin while the next part stands at the stop
		// over it. A cut part waits in the chuck instead, as the real cell does when the line
		// runs dry. A machine with a part finished is served first: it is holding one hostage.
		IF PX_S1 AND AS_S1_UP AND M1_STATE = 2 THEN
			TGT := 0;
			ST1_STEP := 11;
		ELSIF PX_S2 AND AS_S2_UP AND M2_STATE = 2 THEN
			TGT := 1;
			ST1_STEP := 11;
		ELSIF PX_S1 AND AS_S1_UP AND M1_STATE <> 1 THEN
			TGT := 0;
			ST1_STEP := 11;
		ELSIF PX_S2 AND AS_S2_UP AND M2_STATE <> 1 THEN
			TGT := 1;
			ST1_STEP := 11;
		END_IF;
	11:	// over the pin, hand A leading
		GO_POSE := 7;
		GO_RAIL := TGT + 1;
		RX_EXEC := TRUE;
		J1_EXEC := TRUE;
		J2_EXEC := TRUE;
		J3_EXEC := TRUE;
		J4_EXEC := TRUE;
		J5_EXEC := TRUE;
		J6_EXEC := TRUE;
		IF ALL_DONE AND RX_DONE THEN
			ST1_STEP := 12;
		END_IF;
	12:
		J1_EXEC := FALSE;
		J2_EXEC := FALSE;
		J3_EXEC := FALSE;
		J4_EXEC := FALSE;
		J5_EXEC := FALSE;
		J6_EXEC := FALSE;
		RX_EXEC := FALSE;
		// The pin was up with a part on it when this trip was chosen, and the station stays at its
		// ready step until the robot says it is done, so nothing else can have appeared on it. A
		// part that has GONE (the viewer's hand took it) means no exchange: the machine keeps what
		// it has and the watchdog has the last word.
		IF TGT = 0 THEN
			COND := PX_S1;
		ELSE
			COND := PX_S2;
		END_IF;
		IF ALL_CLEAR AND NOT RX_DONE THEN
			IF COND THEN
				ST1_STEP := 13;
			ELSE
				ST1_STEP := 20;
			END_IF;
		END_IF;
	13:	// down onto the pin
		GO_POSE := 6;
		J1_EXEC := TRUE;
		J2_EXEC := TRUE;
		J3_EXEC := TRUE;
		J4_EXEC := TRUE;
		J5_EXEC := TRUE;
		J6_EXEC := TRUE;
		IF ALL_DONE THEN
			ST1_STEP := 14;
		END_IF;
	14:
		J1_EXEC := FALSE;
		J2_EXEC := FALSE;
		J3_EXEC := FALSE;
		J4_EXEC := FALSE;
		J5_EXEC := FALSE;
		J6_EXEC := FALSE;
		IF ALL_CLEAR THEN
			ST1_STEP := 15;
		END_IF;
	15:	// the pin lets go as the fingers close: a hand-over, as out of a chuck
		GRIP_A := TRUE;
		IF T_GRIP.Q AND NOT AS_A_OPEN THEN
			HAS_RAW := TRUE;
			IF TGT = 0 THEN
				S1_CLAMP := FALSE;
			ELSE
				S2_CLAMP := FALSE;
			END_IF;
			ST1_STEP := 16;
		END_IF;
	16:
		GO_POSE := 7;
		J1_EXEC := TRUE;
		J2_EXEC := TRUE;
		J3_EXEC := TRUE;
		J4_EXEC := TRUE;
		J5_EXEC := TRUE;
		J6_EXEC := TRUE;
		IF ALL_DONE THEN
			ST1_STEP := 17;
		END_IF;
	17:
		J1_EXEC := FALSE;
		J2_EXEC := FALSE;
		J3_EXEC := FALSE;
		J4_EXEC := FALSE;
		J5_EXEC := FALSE;
		J6_EXEC := FALSE;
		IF ALL_CLEAR THEN
			ST1_STEP := 20;
		END_IF;
	20:	// in front of the door
		GO_POSE := 3;
		J1_EXEC := TRUE;
		J2_EXEC := TRUE;
		J3_EXEC := TRUE;
		J4_EXEC := TRUE;
		J5_EXEC := TRUE;
		J6_EXEC := TRUE;
		IF ALL_DONE THEN
			ST1_STEP := 21;
		END_IF;
	21:
		J1_EXEC := FALSE;
		J2_EXEC := FALSE;
		J3_EXEC := FALSE;
		J4_EXEC := FALSE;
		J5_EXEC := FALSE;
		J6_EXEC := FALSE;
		IF ALL_CLEAR THEN
			ST1_STEP := 22;
		END_IF;
	22:	// the door must be OPEN before reaching in
		IF TGT = 0 THEN
			SOL_M1_DOOR := TRUE;
			IF AS_M1_DOOR_OP THEN
				ST1_STEP := 23;
			END_IF;
		ELSE
			SOL_M2_DOOR := TRUE;
			IF AS_M2_DOOR_OP THEN
				ST1_STEP := 23;
			END_IF;
		END_IF;
	23:
		IF (TGT = 0 AND M1_STATE = 2) OR (TGT = 1 AND M2_STATE = 2) THEN
			ST1_STEP := 30;
		ELSIF HAS_RAW THEN
			ST1_STEP := 40;
		ELSE
			ST1_STEP := 60;
		END_IF;
	30:	// hand B into the machine, clear of the chuck
		GO_POSE := 5;
		J1_EXEC := TRUE;
		J2_EXEC := TRUE;
		J3_EXEC := TRUE;
		J4_EXEC := TRUE;
		J5_EXEC := TRUE;
		J6_EXEC := TRUE;
		IF ALL_DONE THEN
			ST1_STEP := 31;
		END_IF;
	31:
		J1_EXEC := FALSE;
		J2_EXEC := FALSE;
		J3_EXEC := FALSE;
		J4_EXEC := FALSE;
		J5_EXEC := FALSE;
		J6_EXEC := FALSE;
		IF ALL_CLEAR THEN
			ST1_STEP := 32;
		END_IF;
	32:	// onto the finished part
		GO_POSE := 4;
		J1_EXEC := TRUE;
		J2_EXEC := TRUE;
		J3_EXEC := TRUE;
		J4_EXEC := TRUE;
		J5_EXEC := TRUE;
		J6_EXEC := TRUE;
		IF ALL_DONE THEN
			ST1_STEP := 33;
		END_IF;
	33:
		J1_EXEC := FALSE;
		J2_EXEC := FALSE;
		J3_EXEC := FALSE;
		J4_EXEC := FALSE;
		J5_EXEC := FALSE;
		J6_EXEC := FALSE;
		IF ALL_CLEAR THEN
			ST1_STEP := 34;
		END_IF;
	34:	// grip, then the chuck opens
		GRIP_B := TRUE;
		IF T_GRIP.Q AND NOT AS_B_OPEN THEN
			HAS_FIN := TRUE;
			IF TGT = 0 THEN
				M1_CHUCK := FALSE;
				M1_STATE := 0;
			ELSE
				M2_CHUCK := FALSE;
				M2_STATE := 0;
			END_IF;
			ST1_STEP := 35;
		END_IF;
	35:
		GO_POSE := 5;
		J1_EXEC := TRUE;
		J2_EXEC := TRUE;
		J3_EXEC := TRUE;
		J4_EXEC := TRUE;
		J5_EXEC := TRUE;
		J6_EXEC := TRUE;
		IF ALL_DONE THEN
			ST1_STEP := 36;
		END_IF;
	36:
		J1_EXEC := FALSE;
		J2_EXEC := FALSE;
		J3_EXEC := FALSE;
		J4_EXEC := FALSE;
		J5_EXEC := FALSE;
		J6_EXEC := FALSE;
		IF ALL_CLEAR THEN
			IF HAS_RAW THEN
				ST1_STEP := 40;
			ELSE
				ST1_STEP := 60;
			END_IF;
		END_IF;
	40:	// hand A into the machine, clear of the chuck
		GO_POSE := 2;
		J1_EXEC := TRUE;
		J2_EXEC := TRUE;
		J3_EXEC := TRUE;
		J4_EXEC := TRUE;
		J5_EXEC := TRUE;
		J6_EXEC := TRUE;
		IF ALL_DONE THEN
			ST1_STEP := 41;
		END_IF;
	41:
		J1_EXEC := FALSE;
		J2_EXEC := FALSE;
		J3_EXEC := FALSE;
		J4_EXEC := FALSE;
		J5_EXEC := FALSE;
		J6_EXEC := FALSE;
		IF ALL_CLEAR THEN
			ST1_STEP := 42;
		END_IF;
	42:	// the raw part into the chuck
		GO_POSE := 1;
		J1_EXEC := TRUE;
		J2_EXEC := TRUE;
		J3_EXEC := TRUE;
		J4_EXEC := TRUE;
		J5_EXEC := TRUE;
		J6_EXEC := TRUE;
		IF ALL_DONE THEN
			ST1_STEP := 43;
		END_IF;
	43:
		J1_EXEC := FALSE;
		J2_EXEC := FALSE;
		J3_EXEC := FALSE;
		J4_EXEC := FALSE;
		J5_EXEC := FALSE;
		J6_EXEC := FALSE;
		IF ALL_CLEAR THEN
			ST1_STEP := 44;
		END_IF;
	44:	// the chuck closes, the hand opens, the cut starts
		GRIP_A := FALSE;
		IF TGT = 0 THEN
			M1_CHUCK := TRUE;
		ELSE
			M2_CHUCK := TRUE;
		END_IF;
		IF T_GRIP.Q AND AS_A_OPEN THEN
			HAS_RAW := FALSE;
			IF TGT = 0 THEN
				M1_STATE := 1;
			ELSE
				M2_STATE := 1;
			END_IF;
			ST1_STEP := 45;
		END_IF;
	45:
		GO_POSE := 2;
		J1_EXEC := TRUE;
		J2_EXEC := TRUE;
		J3_EXEC := TRUE;
		J4_EXEC := TRUE;
		J5_EXEC := TRUE;
		J6_EXEC := TRUE;
		IF ALL_DONE THEN
			ST1_STEP := 46;
		END_IF;
	46:
		J1_EXEC := FALSE;
		J2_EXEC := FALSE;
		J3_EXEC := FALSE;
		J4_EXEC := FALSE;
		J5_EXEC := FALSE;
		J6_EXEC := FALSE;
		IF ALL_CLEAR THEN
			ST1_STEP := 60;
		END_IF;
	60:	// out of the machine
		GO_POSE := 3;
		J1_EXEC := TRUE;
		J2_EXEC := TRUE;
		J3_EXEC := TRUE;
		J4_EXEC := TRUE;
		J5_EXEC := TRUE;
		J6_EXEC := TRUE;
		IF ALL_DONE THEN
			ST1_STEP := 61;
		END_IF;
	61:
		J1_EXEC := FALSE;
		J2_EXEC := FALSE;
		J3_EXEC := FALSE;
		J4_EXEC := FALSE;
		J5_EXEC := FALSE;
		J6_EXEC := FALSE;
		IF ALL_CLEAR THEN
			ST1_STEP := 62;
		END_IF;
	62:	// shut the door on the cut
		IF TGT = 0 THEN
			SOL_M1_DOOR := FALSE;
			COND := AS_M1_DOOR_CL;
		ELSE
			SOL_M2_DOOR := FALSE;
			COND := AS_M2_DOOR_CL;
		END_IF;
		IF COND THEN
			IF HAS_FIN THEN
				ST1_STEP := 70;
			ELSE
				ST1_STEP := 80;
			END_IF;
		END_IF;
	70:	// hand B over the pin the part came off
		GO_POSE := 9;
		J1_EXEC := TRUE;
		J2_EXEC := TRUE;
		J3_EXEC := TRUE;
		J4_EXEC := TRUE;
		J5_EXEC := TRUE;
		J6_EXEC := TRUE;
		IF ALL_DONE THEN
			ST1_STEP := 71;
		END_IF;
	71:
		J1_EXEC := FALSE;
		J2_EXEC := FALSE;
		J3_EXEC := FALSE;
		J4_EXEC := FALSE;
		J5_EXEC := FALSE;
		J6_EXEC := FALSE;
		IF ALL_CLEAR THEN
			ST1_STEP := 72;
		END_IF;
	72:
		GO_POSE := 8;
		J1_EXEC := TRUE;
		J2_EXEC := TRUE;
		J3_EXEC := TRUE;
		J4_EXEC := TRUE;
		J5_EXEC := TRUE;
		J6_EXEC := TRUE;
		IF ALL_DONE THEN
			ST1_STEP := 73;
		END_IF;
	73:
		J1_EXEC := FALSE;
		J2_EXEC := FALSE;
		J3_EXEC := FALSE;
		J4_EXEC := FALSE;
		J5_EXEC := FALSE;
		J6_EXEC := FALSE;
		IF ALL_CLEAR THEN
			ST1_STEP := 74;
		END_IF;
	74:	// the pin takes it, the hand lets go
		GRIP_B := FALSE;
		IF TGT = 0 THEN
			S1_CLAMP := TRUE;
			COND := PX_S1;
		ELSE
			S2_CLAMP := TRUE;
			COND := PX_S2;
		END_IF;
		IF T_GRIP.Q AND AS_B_OPEN AND COND THEN
			HAS_FIN := FALSE;
			ST1_STEP := 75;
		END_IF;
	75:
		GO_POSE := 9;
		J1_EXEC := TRUE;
		J2_EXEC := TRUE;
		J3_EXEC := TRUE;
		J4_EXEC := TRUE;
		J5_EXEC := TRUE;
		J6_EXEC := TRUE;
		IF ALL_DONE THEN
			ST1_STEP := 76;
		END_IF;
	76:
		J1_EXEC := FALSE;
		J2_EXEC := FALSE;
		J3_EXEC := FALSE;
		J4_EXEC := FALSE;
		J5_EXEC := FALSE;
		J6_EXEC := FALSE;
		IF ALL_CLEAR THEN
			ST1_STEP := 80;
		END_IF;
	80:	// done at this station: the pin may go down and the station is free again
		IF TGT = 0 THEN
			S1_GO := TRUE;
		ELSE
			S2_GO := TRUE;
		END_IF;
		CYCLE_CNT := CYCLE_CNT + 1;
		IF STOP_REQ THEN
			ST1_STEP := 0;
		ELSE
			ST1_STEP := 10;
		END_IF;
	800:	// HOME: the arm to its travel pose over machine 1
		EM_IN_EMIT := FALSE;
		CV_RUN := FALSE;
		SOL_M1_DOOR := FALSE;
		SOL_M2_DOOR := FALSE;
		GO_POSE := 10;
		GO_RAIL := 1;
		RX_EXEC := TRUE;
		J1_EXEC := TRUE;
		J2_EXEC := TRUE;
		J3_EXEC := TRUE;
		J4_EXEC := TRUE;
		J5_EXEC := TRUE;
		J6_EXEC := TRUE;
		IF ALL_DONE AND RX_DONE THEN
			J1_EXEC := FALSE;
			J2_EXEC := FALSE;
			J3_EXEC := FALSE;
			J4_EXEC := FALSE;
			J5_EXEC := FALSE;
			J6_EXEC := FALSE;
			RX_EXEC := FALSE;
			HOMED := TRUE;
			ST1_STEP := 0;
		END_IF;
	900:	// stuck, or the selector was turned while running
		J1_EXEC := FALSE;
		J2_EXEC := FALSE;
		J3_EXEC := FALSE;
		J4_EXEC := FALSE;
		J5_EXEC := FALSE;
		J6_EXEC := FALSE;
		RX_EXEC := FALSE;
		EM_IN_EMIT := FALSE;
		CV_RUN := FALSE;
		IF START_EDGE AND SEL_AUTO THEN
			STOP_REQ := FALSE;
			ST1_STEP := 0;
		END_IF;
	910:	// the master circuit is open: the jaws, the chucks and the pins KEEP what they hold
		J1_EXEC := FALSE;
		J2_EXEC := FALSE;
		J3_EXEC := FALSE;
		J4_EXEC := FALSE;
		J5_EXEC := FALSE;
		J6_EXEC := FALSE;
		RX_EXEC := FALSE;
		EM_IN_EMIT := FALSE;
		CV_RUN := FALSE;
		IF READY THEN
			ST1_STEP := 0;
		END_IF;
END_CASE;

RUNNING := ST1_STEP <> 0 AND ST1_STEP <> 800 AND ST1_STEP <> 900 AND ST1_STEP <> 910;
IF RUNNING THEN
	CV_RUN := TRUE;
END_IF;

// ---------------------------------------------------------- ST2: machine 1, the cut
IF NOT RUNNING THEN
	ST2_STEP := 0;
ELSE
	CASE ST2_STEP OF
		100:
			IF M1_STATE = 1 THEN
				ST2_STEP := 110;
			END_IF;
		110:	// the door stays shut and the chuck stays closed for the whole of it
			IF T_CUT1.Q THEN
				M1_STATE := 2;
				ST2_STEP := 120;
			END_IF;
		120:	// the robot has taken it
			IF M1_STATE <> 2 THEN
				ST2_STEP := 100;
			END_IF;
	ELSE
		ST2_STEP := 100;
	END_CASE;
END_IF;

// ---------------------------------------------------------- ST3: machine 2, the cut
IF NOT RUNNING THEN
	ST3_STEP := 0;
ELSE
	CASE ST3_STEP OF
		100:
			IF M2_STATE = 1 THEN
				ST3_STEP := 110;
			END_IF;
		110:
			IF T_CUT2.Q THEN
				M2_STATE := 2;
				ST3_STEP := 120;
			END_IF;
		120:
			IF M2_STATE <> 2 THEN
				ST3_STEP := 100;
			END_IF;
	ELSE
		ST3_STEP := 100;
	END_CASE;
END_IF;

// ---------------------------------------------------------- ST4: station 1 and the feed
IF NOT RUNNING THEN
	ST4_STEP := 0;
	EM_IN_EMIT := FALSE;
ELSE
	CASE ST4_STEP OF
		200:	// down, stop up, nothing on the pin: call for one raw part
			SOL_S1_UP := FALSE;
			SOL_S1_DN := TRUE;
			SOL_S1_STOP := TRUE;
			S1_CLAMP := FALSE;
			S1_GO := FALSE;
			IF AS_S1_STOP_UP AND NOT PE_S1 THEN
				EM_IN_EMIT := TRUE;
				ST4_STEP := 210;
			END_IF;
		210:
			EM_IN_EMIT := FALSE;
			IF PE_S1 THEN
				ST4_STEP := 220;
			END_IF;
		220:	// the beam says the part is HERE; the STOP is what locates it, so keep driving
			IF T_SETTLE1.Q THEN
				SOL_S1_DN := FALSE;
				SOL_S1_UP := TRUE;
				S1_CLAMP := TRUE;
				ST4_STEP := 230;
			END_IF;
		230:
			IF AS_S1_UP THEN
				ST4_STEP := 240;
			END_IF;
		240:	// ready for the robot, and waiting for it to finish at this station
			IF S1_GO THEN
				S1_GO := FALSE;
				IF PX_S1 THEN
					ST4_STEP := 250;
				ELSE
					ST4_STEP := 270;
				END_IF;
			END_IF;
		250:	// let go FIRST, so the part rides the pin down and the pin drops away under it
			S1_CLAMP := FALSE;
			IF T_DROP1.Q THEN
				ST4_STEP := 260;
			END_IF;
		260:	// the STOP goes down BEFORE the pin: with it still up the part comes down onto the
			// 30 mm stop head instead of the belt, stands on its rim and topples. Station 2 must
			// be empty and clear too: two parts at one stop cannot be metered apart again.
			IF ST5_STEP = 200 AND NOT PE_S2 THEN
				SOL_S1_STOP := FALSE;
				ST4_STEP := 262;
			END_IF;
		262:
			IF AS_S1_STOP_DN THEN
				SOL_S1_UP := FALSE;
				SOL_S1_DN := TRUE;
				ST4_STEP := 265;
			END_IF;
		265:
			IF AS_S1_DN AND NOT PE_S1 THEN
				SOL_S1_STOP := TRUE;
				ST4_STEP := 200;
			END_IF;
		270:
			S1_CLAMP := FALSE;
			SOL_S1_UP := FALSE;
			SOL_S1_DN := TRUE;
			IF AS_S1_DN THEN
				ST4_STEP := 200;
			END_IF;
	ELSE
		ST4_STEP := 200;
	END_CASE;
END_IF;

// ---------------------------------------------------------- ST5: station 2 and the discharge
IF NOT RUNNING THEN
	ST5_STEP := 0;
ELSE
	CASE ST5_STEP OF
		200:
			SOL_S2_UP := FALSE;
			SOL_S2_DN := TRUE;
			SOL_S2_STOP := TRUE;
			S2_CLAMP := FALSE;
			S2_GO := FALSE;
			IF PE_S2 THEN
				ST5_STEP := 220;
			END_IF;
		220:
			IF T_SETTLE2.Q THEN
				SOL_S2_DN := FALSE;
				SOL_S2_UP := TRUE;
				S2_CLAMP := TRUE;
				ST5_STEP := 230;
			END_IF;
		230:
			IF AS_S2_UP THEN
				ST5_STEP := 240;
			END_IF;
		240:
			IF S2_GO THEN
				S2_GO := FALSE;
				IF PX_S2 THEN
					ST5_STEP := 250;
				ELSE
					ST5_STEP := 270;
				END_IF;
			END_IF;
		250:
			S2_CLAMP := FALSE;
			IF T_DROP2.Q THEN
				ST5_STEP := 260;
			END_IF;
		260:
			SOL_S2_STOP := FALSE;
			ST5_STEP := 262;
		262:
			IF AS_S2_STOP_DN THEN
				SOL_S2_UP := FALSE;
				SOL_S2_DN := TRUE;
				ST5_STEP := 265;
			END_IF;
		265:
			IF AS_S2_DN AND NOT PE_S2 THEN
				SOL_S2_STOP := TRUE;
				ST5_STEP := 200;
			END_IF;
		270:
			S2_CLAMP := FALSE;
			SOL_S2_UP := FALSE;
			SOL_S2_DN := TRUE;
			IF AS_S2_DN THEN
				ST5_STEP := 200;
			END_IF;
	ELSE
		ST5_STEP := 200;
	END_CASE;
END_IF;

// The joint targets for the pose the step asked for. GENERATED - see the header.
// BEGIN GENERATED - tools/gen_lathe_line.js
CASE GO_POSE OF
	1:	// chAtA
		J1_TGT := -93.18;
		J2_TGT := 7.66;
		J3_TGT := -37.91;
		J4_TGT := 91.60;
		J5_TGT := -87.24;
		J6_TGT := 0.00;
	2:	// chOutA
		J1_TGT := -74.48;
		J2_TGT := 10.03;
		J3_TGT := -40.73;
		J4_TGT := 81.92;
		J5_TGT := -103.29;
		J6_TGT := 0.00;
	3:	// doorA
		J1_TGT := -124.77;
		J2_TGT := -54.34;
		J3_TGT := -17.86;
		J4_TGT := 123.46;
		J5_TGT := -79.95;
		J6_TGT := 0.00;
	4:	// chAtB
		J1_TGT := -108.80;
		J2_TGT := -1.09;
		J3_TGT := -12.69;
		J4_TGT := -7.37;
		J5_TGT := -57.72;
		J6_TGT := 111.71;
	5:	// chOutB
		J1_TGT := -88.59;
		J2_TGT := -4.61;
		J3_TGT := -9.64;
		J4_TGT := 0.66;
		J5_TGT := -53.28;
		J6_TGT := 88.31;
	6:	// pinAtA
		J1_TGT := 66.86;
		J2_TGT := -42.35;
		J3_TGT := 8.50;
		J4_TGT := 0.01;
		J5_TGT := -56.15;
		J6_TGT := 0.00;
	7:	// pinUpA
		J1_TGT := 66.82;
		J2_TGT := -51.18;
		J3_TGT := 29.70;
		J4_TGT := 0.00;
		J5_TGT := -68.51;
		J6_TGT := 0.00;
	8:	// pinAtB
		J1_TGT := 71.46;
		J2_TGT := -41.47;
		J3_TGT := -14.24;
		J4_TGT := -3.70;
		J5_TGT := 55.75;
		J6_TGT := 2.09;
	9:	// pinUpB
		J1_TGT := 71.08;
		J2_TGT := -54.82;
		J3_TGT := 10.71;
		J4_TGT := -4.03;
		J5_TGT := 44.19;
		J6_TGT := 2.90;
	10:	// home
		J1_TGT := 4.43;
		J2_TGT := -47.26;
		J3_TGT := 42.85;
		J4_TGT := 0.01;
		J5_TGT := -85.59;
		J6_TGT := 0.00;
END_CASE;
CASE GO_RAIL OF
	1:	RX_TGT := -980.00;
	2:	RX_TGT := 620.00;
END_CASE;
// END GENERATED

// TONs after the CASE: their Q is read by the NEXT scan.
T_GRIP(In := ST1_STEP = 15 OR ST1_STEP = 34 OR ST1_STEP = 44 OR ST1_STEP = 74, PT := T#400ms);
T_SETTLE1(In := ST4_STEP = 220, PT := T#700ms);
T_SETTLE2(In := ST5_STEP = 220, PT := T#700ms);
T_DROP1(In := ST4_STEP = 250, PT := T#200ms);
T_DROP2(In := ST5_STEP = 250, PT := T#200ms);
T_CUT1(In := M1_STATE = 1, PT := T#20s);
T_CUT2(In := M2_STATE = 1, PT := T#20s);

// Watchdog: a running step that stops moving is a jam, not patience. A station that stops moving
// is one too - a part taken off the belt by hand leaves one waiting for a beam that never comes,
// and a machine that waits for ever looks alive.
// The TON is called BEFORE STEP_LAST is updated, so a step change gives it one scan of In = FALSE
// and resets it. Updating first would make the compare always true and the watchdog never reset.
T_WD(In := ST1_STEP <> 0 AND ST1_STEP <> 900 AND ST1_STEP <> 910 AND ST1_STEP = STEP_LAST, PT := T#45s);
STEP_LAST := ST1_STEP;
// Only the station steps that MOVE something are watched. The ones that wait for the line - for a
// part to be sent on (200, 210) and for the robot (240) - are not jams: the robot is 45 s away
// whenever it stands over the other machine through a 20 s cut.
T_WD4(In := RUNNING AND ST4_STEP >= 220 AND ST4_STEP <> 240, PT := T#45s);
T_WD5(In := RUNNING AND ST5_STEP >= 220 AND ST5_STEP <> 240, PT := T#45s);
IF T_WD.Q OR T_WD4.Q OR T_WD5.Q OR (SEL_CHANGED AND RUNNING) THEN
	ST1_STEP := 900;
	J1_EXEC := FALSE;
	J2_EXEC := FALSE;
	J3_EXEC := FALSE;
	J4_EXEC := FALSE;
	J5_EXEC := FALSE;
	J6_EXEC := FALSE;
	RX_EXEC := FALSE;
	EM_IN_EMIT := FALSE;
	CV_RUN := FALSE;
END_IF;

IF ESTOP THEN
	IF ST1_STEP <> 910 THEN
		ST1_STEP := 910;
	END_IF;
	J1_EXEC := FALSE;
	J2_EXEC := FALSE;
	J3_EXEC := FALSE;
	J4_EXEC := FALSE;
	J5_EXEC := FALSE;
	J6_EXEC := FALSE;
	RX_EXEC := FALSE;
	EM_IN_EMIT := FALSE;
	CV_RUN := FALSE;
ELSIF HOME_EDGE AND READY AND ST1_STEP = 0 THEN
	ST1_STEP := 800;
END_IF;

AUTO_RUN := ST1_STEP <> 0 AND ST1_STEP <> 800 AND ST1_STEP <> 900 AND ST1_STEP <> 910;
IND_ACTIVE := NOT SEL_AUTO AND NOT AUTO_RUN AND READY AND ST1_STEP <> 800;
IF IND_ACTIVE THEN
	IF IND_A AND NOT IND_A_LAST THEN
		MEM_A := NOT MEM_A;
	END_IF;
	IF IND_B AND NOT IND_B_LAST THEN
		MEM_B := NOT MEM_B;
	END_IF;
	IF IND_DOOR1 AND NOT IND_D1_LAST THEN
		MEM_D1 := NOT MEM_D1;
	END_IF;
	IF IND_DOOR2 AND NOT IND_D2_LAST THEN
		MEM_D2 := NOT MEM_D2;
	END_IF;
	IF IND_LIFT1 AND NOT IND_L1_LAST THEN
		MEM_L1 := NOT MEM_L1;
	END_IF;
	IF IND_LIFT2 AND NOT IND_L2_LAST THEN
		MEM_L2 := NOT MEM_L2;
	END_IF;
	GRIP_A := MEM_A;
	GRIP_B := MEM_B;
	SOL_M1_DOOR := MEM_D1;
	SOL_M2_DOOR := MEM_D2;
	SOL_S1_UP := MEM_L1;
	SOL_S1_DN := NOT MEM_L1;
	SOL_S2_UP := MEM_L2;
	SOL_S2_DN := NOT MEM_L2;
ELSE
	MEM_A := FALSE;
	MEM_B := FALSE;
	MEM_D1 := FALSE;
	MEM_D2 := FALSE;
	MEM_L1 := FALSE;
	MEM_L2 := FALSE;
END_IF;
IND_A_LAST := IND_A;
IND_B_LAST := IND_B;
IND_D1_LAST := IND_DOOR1;
IND_D2_LAST := IND_DOOR2;
IND_L1_LAST := IND_LIFT1;
IND_L2_LAST := IND_LIFT2;
J1_JOG_P := IND_ACTIVE AND IND_J1_P;
J1_JOG_N := IND_ACTIVE AND IND_J1_N;
J2_JOG_P := IND_ACTIVE AND IND_J2_P;
J2_JOG_N := IND_ACTIVE AND IND_J2_N;
J3_JOG_P := IND_ACTIVE AND IND_J3_P;
J3_JOG_N := IND_ACTIVE AND IND_J3_N;
J4_JOG_P := IND_ACTIVE AND IND_J4_P;
J4_JOG_N := IND_ACTIVE AND IND_J4_N;
J5_JOG_P := IND_ACTIVE AND IND_J5_P;
J5_JOG_N := IND_ACTIVE AND IND_J5_N;
J6_JOG_P := IND_ACTIVE AND IND_J6_P;
J6_JOG_N := IND_ACTIVE AND IND_J6_N;
RX_JOG_P := IND_ACTIVE AND IND_RX_P;
RX_JOG_N := IND_ACTIVE AND IND_RX_N;

OVR := OVR_SET;
PL_START := AUTO_RUN;
PL_MASTER := MASTER_ON;
PL_HOME := HOMED;
